LIN {X 0,Y 411.182,Z 344.267,A -85,B 0,C 180,E1 -10470.848,E2 -10470.848} C_VEL
LIN {X 0,Y 411.197,Z 344.265,A -85,B 0,C 180,E1 -10474.334,E2 -10474.334} C_VEL
LIN {X 0,Y 411.18,Z 344.267,A -85,B 0,C 180,E1 -10477.975,E2 -10477.975} C_VEL
LIN {X 0,Y 411.141,Z 344.272,A -85,B 0,C 180,E1 -10481.226,E2 -10481.226} C_VEL
LIN {X 0,Y 411.169,Z 344.265,A -85,B 0,C 180,E1 -10484.492,E2 -10484.492} C_VEL
LIN {X 0,Y 411.213,Z 344.444,A -85,B 0,C 180,E1 -10487.137,E2 -10487.137} C_VEL
LIN {X 0,Y 412.973,Z 353.126,A -85,B 0,C 180,E1 -10490.516,E2 -10490.516} C_VEL
LIN {X 0,Y 414.178,Z 359.884,A -85,B 0,C 180,E1 -10492.894,E2 -10492.894} C_VEL
LIN {X 0,Y 413.948,Z 363.821,A -85,B 0,C 180,E1 -10494.146,E2 -10494.146} C_VEL
LIN {X 0,Y 412.826,Z 377.183,A -85,B 0,C 180,E1 -10498.147,E2 -10498.147} C_VEL
LIN {X 0,Y 412.116,Z 388.901,A -85,B 0,C 180,E1 -10501.479,E2 -10501.479} C_VEL
LIN {X 0,Y 411.506,Z 401.226,A -85,B 0,C 180,E1 -10504.847,E2 -10504.847} C_VEL
LIN {X 0,Y 411.04,Z 414.75,A -85,B 0,C 180,E1 -10508.432,E2 -10508.432} C_VEL
LIN {X 0,Y 410.751,Z 427.741,A -85,B 0,C 180,E1 -10511.805,E2 -10511.805} C_VEL
LIN {X 0,Y 410.736,Z 429.149,A -85,B 0,C 180,E1 -10512.091,E2 -10512.091} C_VEL
LIN {X 0,Y 412.704,Z 446.705,A -85,B 0,C 180,E1 -10512.79,E2 -10512.79} C_VEL
LIN {X 0,Y 413.305,Z 460.605,A -85,B 0,C 180,E1 -10513.516,E2 -10513.516} C_VEL
LIN {X 0,Y 413.672,Z 472.997,A -85,B 0,C 180,E1 -10514.354,E2 -10514.354} C_VEL
LIN {X 0,Y 412.741,Z 484.841,A -85,B 0,C 180,E1 -10515.328,E2 -10515.328} C_VEL
LIN {X 0,Y 411.972,Z 495.807,A -85,B 0,C 180,E1 -10516.46,E2 -10516.46} C_VEL
LIN {X 0,Y 411.62,Z 503.6,A -85,B 0,C 180,E1 -10517.427,E2 -10517.427} C_VEL
LIN {X 0,Y 411.044,Z 512.023,A -85,B 0,C 180,E1 -10518.661,E2 -10518.661} C_VEL
LIN {X 0,Y 410.621,Z 520.378,A -85,B 0,C 180,E1 -10520.145,E2 -10520.145} C_VEL
LIN {X 0,Y 410.458,Z 527.159,A -85,B 0,C 180,E1 -10521.632,E2 -10521.632} C_VEL
LIN {X 0,Y 410.452,Z 533.082,A -85,B 0,C 180,E1 -10523.272,E2 -10523.272} C_VEL
LIN {X 0,Y 410.58,Z 538.034,A -85,B 0,C 180,E1 -10525.09,E2 -10525.09} C_VEL
LIN {X 0,Y 410.673,Z 540.042,A -85,B 0,C 180,E1 -10526.075,E2 -10526.075} C_VEL
LIN {X 0,Y 410.66,Z 542.668,A -85,B 0,C 180,E1 -10528.039,E2 -10528.039} C_VEL
LIN {X 0,Y 410.893,Z 543.399,A -85,B 0,C 180,E1 -10529.02,E2 -10529.02} C_VEL
LIN {X 0,Y 410.904,Z 543.637,A -85,B 0,C 180,E1 -10530,E2 -10530} C_VEL
LIN {X 0,Y 410.886,Z 543.448,A -85,B 0,C 180,E1 -10530.98,E2 -10530.98} C_VEL
LIN {X 0,Y 410.614,Z 541.808,A -85,B 0,C 180,E1 -10532.943,E2 -10532.943} C_VEL
LIN {X 0,Y 410.637,Z 540.321,A -85,B 0,C 180,E1 -10533.925,E2 -10533.925} C_VEL
LIN {X 0,Y 410.505,Z 537.236,A -85,B 0,C 180,E1 -10535.403,E2 -10535.403} C_VEL
LIN {X 0,Y 410.458,Z 533.052,A -85,B 0,C 180,E1 -10536.884,E2 -10536.884} C_VEL
LIN {X 0,Y 410.472,Z 526.635,A -85,B 0,C 180,E1 -10538.616,E2 -10538.616} C_VEL
LIN {X 0,Y 410.643,Z 519.625,A -85,B 0,C 180,E1 -10540.103,E2 -10540.103} C_VEL
LIN {X 0,Y 411.109,Z 510.866,A -85,B 0,C 180,E1 -10541.587,E2 -10541.587} C_VEL
LIN {X 0,Y 411.758,Z 500.837,A -85,B 0,C 180,E1 -10542.962,E2 -10542.962} C_VEL
LIN {X 0,Y 412.365,Z 490.938,A -85,B 0,C 180,E1 -10544.055,E2 -10544.055} C_VEL
LIN {X 0,Y 413.044,Z 479.935,A -85,B 0,C 180,E1 -10545.039,E2 -10545.039} C_VEL
LIN {X 0,Y 413.6,Z 469.683,A -85,B 0,C 180,E1 -10545.776,E2 -10545.776} C_VEL
LIN {X 0,Y 412.83,Z 456.929,A -85,B 0,C 180,E1 -10546.527,E2 -10546.527} C_VEL
LIN {X 0,Y 411.742,Z 444.07,A -85,B 0,C 180,E1 -10547.086,E2 -10547.086} C_VEL
LIN {X 0,Y 410.691,Z 433.86,A -85,B 0,C 180,E1 -10547.445,E2 -10547.445} C_VEL
LIN {X 0,Y 411.003,Z 424.02,A -85,B 0,C 180,E1 -10549.998,E2 -10549.998} C_VEL
LIN {X 0,Y 411.592,Z 410.426,A -85,B 0,C 180,E1 -10553.657,E2 -10553.657} C_VEL
LIN {X 0,Y 412.186,Z 398.684,A -85,B 0,C 180,E1 -10556.861,E2 -10556.861} C_VEL
LIN {X 0,Y 413.082,Z 384.959,A -85,B 0,C 180,E1 -10560.69,E2 -10560.69} C_VEL
LIN {X 0,Y 413.961,Z 373.104,A -85,B 0,C 180,E1 -10564.072,E2 -10564.072} C_VEL
LIN {X 0,Y 414.818,Z 363.878,A -85,B 0,C 180,E1 -10566.78,E2 -10566.78} C_VEL
LIN {X 0,Y 413.734,Z 357.047,A -85,B 0,C 180,E1 -10568.939,E2 -10568.939} C_VEL
LIN {X 0,Y 411.767,Z 347.244,A -85,B 0,C 180,E1 -10572.215,E2 -10572.215} C_VEL
LIN {X 0,Y 411.186,Z 344.328,A -85,B 0,C 180,E1 -10573.299,E2 -10573.299} C_VEL
LIN {X 0,Y 411.159,Z 344.271,A -85,B 0,C 180,E1 -10576.864,E2 -10576.864} C_VEL
LIN {X 0,Y 411.163,Z 344.265,A -85,B 0,C 180,E1 -10580.279,E2 -10580.279} C_VEL
LIN {X 0,Y 411.186,Z 344.268,A -85,B 0,C 180,E1 -10583.447,E2 -10583.447} C_VEL
LIN {X 0,Y 411.2,Z 344.263,A -85,B 0,C 180,E1 -10586.873,E2 -10586.873} C_VEL
LIN {X 0,Y 411.225,Z 344.258,A -85,B 0,C 180,E1 -10590.644,E2 -10590.644} C_VEL
LIN {X 0,Y 411.229,Z 344.259,A -85,B 0,C 180,E1 -10593.618,E2 -10593.618} C_VEL
LIN {X 0,Y 411.187,Z 344.266,A -85,B 0,C 180,E1 -10596.851,E2 -10596.851} C_VEL
LIN {X 0,Y 411.205,Z 344.259,A -85,B 0,C 180,E1 -10600.05,E2 -10600.05} C_VEL
LIN {X 0,Y 411.254,Z 344.26,A -85,B 0,C 180,E1 -10603.131,E2 -10603.131} C_VEL
LIN {X 0,Y 411.296,Z 344.254,A -85,B 0,C 180,E1 -10606.896,E2 -10606.896} C_VEL
LIN {X 0,Y 411.281,Z 344.25,A -85,B 0,C 180,E1 -10610.161,E2 -10610.161} C_VEL
LIN {X 0,Y 411.426,Z 344.236,A -85,B 0,C 180,E1 -10613.132,E2 -10613.132} C_VEL
LIN {X 0,Y 411.296,Z 344.253,A -85,B 0,C 180,E1 -10615.099,E2 -10615.099} C_VEL
LIN {X 0,Y 411.501,Z 344.223,A -85,B 0,C 180,E1 -10618.042,E2 -10618.042} C_VEL
LIN {X 0,Y 411.631,Z 344.207,A -85,B 0,C 180,E1 -10620,E2 -10620} C_VEL
LIN {X 0,Y 411.446,Z 344.235,A -85,B 0,C 180,E1 -10622.937,E2 -10622.937} C_VEL
LIN {X 0,Y 411.448,Z 344.234,A -85,B 0,C 180,E1 -10626.867,E2 -10626.867} C_VEL
LIN {X 0,Y 411.284,Z 344.25,A -85,B 0,C 180,E1 -10629.839,E2 -10629.839} C_VEL
LIN {X 0,Y 411.296,Z 344.25,A -85,B 0,C 180,E1 -10633.104,E2 -10633.104} C_VEL
LIN {X 0,Y 411.249,Z 344.257,A -85,B 0,C 180,E1 -10636.889,E2 -10636.889} C_VEL
LIN {X 0,Y 411.222,Z 344.259,A -85,B 0,C 180,E1 -10639.987,E2 -10639.987} C_VEL
LIN {X 0,Y 411.196,Z 344.261,A -85,B 0,C 180,E1 -10643.148,E2 -10643.148} C_VEL
LIN {X 0,Y 411.23,Z 344.263,A -85,B 0,C 180,E1 -10646.381,E2 -10646.381} C_VEL
LIN {X 0,Y 411.203,Z 344.26,A -85,B 0,C 180,E1 -10649.713,E2 -10649.713} C_VEL
LIN {X 0,Y 411.2,Z 344.26,A -85,B 0,C 180,E1 -10653.156,E2 -10653.156} C_VEL
LIN {X 0,Y 411.189,Z 344.265,A -85,B 0,C 180,E1 -10656.554,E2 -10656.554} C_VEL
LIN {X 0,Y 411.221,Z 344.259,A -85,B 0,C 180,E1 -10659.731,E2 -10659.731} C_VEL
LIN {X 0,Y 411.172,Z 344.263,A -85,B 0,C 180,E1 -10663.134,E2 -10663.134} C_VEL
LIN {X 0,Y 411.169,Z 344.268,A -85,B 0,C 180,E1 -10665.881,E2 -10665.881} C_VEL
LIN {X 0,Y 411.165,Z 344.265,A -85,B 0,C 180,E1 -10668.772,E2 -10668.772} C_VEL
LIN {X 0,Y 411.208,Z 344.263,A -85,B 0,C 180,E1 -10671.831,E2 -10671.831} C_VEL
LIN {X 0,Y 411.209,Z 344.259,A -85,B 0,C 180,E1 -10675.122,E2 -10675.122} C_VEL
LIN {X 0,Y 411.17,Z 344.271,A -85,B 0,C 180,E1 -10678.004,E2 -10678.004} C_VEL
LIN {X 0,Y 411.223,Z 344.259,A -85,B 0,C 180,E1 -10681.411,E2 -10681.411} C_VEL
LIN {X 0,Y 411.236,Z 344.256,A -85,B 0,C 180,E1 -10684.708,E2 -10684.708} C_VEL
LIN {X 0,Y 411.206,Z 344.266,A -85,B 0,C 180,E1 -10687.914,E2 -10687.914} C_VEL
LIN {X 0,Y 411.226,Z 344.257,A -85,B 0,C 180,E1 -10691.052,E2 -10691.052} C_VEL
LIN {X 0,Y 411.265,Z 344.255,A -85,B 0,C 180,E1 -10694.133,E2 -10694.133} C_VEL
LIN {X 0,Y 411.305,Z 344.248,A -85,B 0,C 180,E1 -10697.166,E2 -10697.166} C_VEL
LIN {X 0,Y 411.296,Z 344.25,A -85,B 0,C 180,E1 -10700.162,E2 -10700.162} C_VEL
LIN {X 0,Y 411.464,Z 344.229,A -85,B 0,C 180,E1 -10703.133,E2 -10703.133} C_VEL
LIN {X 0,Y 411.315,Z 344.248,A -85,B 0,C 180,E1 -10705.099,E2 -10705.099} C_VEL
LIN {X 0,Y 411.516,Z 344.223,A -85,B 0,C 180,E1 -10708.043,E2 -10708.043} C_VEL
LIN {X 0,Y 411.645,Z 344.207,A -85,B 0,C 180,E1 -10710,E2 -10710} C_VEL
LIN {X 0,Y 411.469,Z 344.228,A -85,B 0,C 180,E1 -10712.937,E2 -10712.937} C_VEL
LIN {X 0,Y 411.454,Z 344.23,A -85,B 0,C 180,E1 -10716.867,E2 -10716.867} C_VEL
LIN {X 0,Y 411.295,Z 344.251,A -85,B 0,C 180,E1 -10719.838,E2 -10719.838} C_VEL
LIN {X 0,Y 411.284,Z 344.252,A -85,B 0,C 180,E1 -10723.338,E2 -10723.338} C_VEL
LIN {X 0,Y 411.258,Z 344.255,A -85,B 0,C 180,E1 -10726.888,E2 -10726.888} C_VEL
LIN {X 0,Y 411.241,Z 344.255,A -85,B 0,C 180,E1 -10727.603,E2 -10727.603} C_VEL
LIN {X 0,Y 410.582,Z 344.339,A -85,B 0,C 180,E1 -10728.421,E2 -10728.421} C_VEL
LIN {X 0,Y 407.694,Z 344.702,A -85,B 0,C 180,E1 -10729.749,E2 -10729.749} C_VEL
LIN {X 0,Y 405.249,Z 345.006,A -85,B 0,C 180,E1 -10730.822,E2 -10730.822} C_VEL
LIN {X 0,Y 404.213,Z 345.134,A -85,B 0,C 180,E1 -10731.652,E2 -10731.652} C_VEL
LIN {X 0,Y 404.137,Z 345.141,A -85,B 0,C 180,E1 -10731.933,E2 -10731.933} C_VEL
LIN {X 0,Y 404.216,Z 345.136,A -85,B 0,C 180,E1 -10735.296,E2 -10735.296} C_VEL
LIN {X 0,Y 404.195,Z 345.133,A -85,B 0,C 180,E1 -10737.999,E2 -10737.999} C_VEL
LIN {X 0,Y 404.138,Z 345.142,A -85,B 0,C 180,E1 -10741.557,E2 -10741.557} C_VEL
LIN {X 0,Y 404.184,Z 345.141,A -85,B 0,C 180,E1 -10745.015,E2 -10745.015} C_VEL
LIN {X 0,Y 404.162,Z 345.141,A -85,B 0,C 180,E1 -10748.755,E2 -10748.755} C_VEL
LIN {X 0,Y 404.188,Z 345.138,A -85,B 0,C 180,E1 -10751.61,E2 -10751.61} C_VEL
LIN {X 0,Y 404.209,Z 345.153,A -85,B 0,C 180,E1 -10755.21,E2 -10755.21} C_VEL
LIN {X 0,Y 404.325,Z 345.754,A -85,B 0,C 180,E1 -10755.451,E2 -10755.451} C_VEL
LIN {X 0,Y 408.011,Z 358.828,A -85,B 0,C 180,E1 -10756.499,E2 -10756.499} C_VEL
LIN {X 0,Y 408.323,Z 361.622,A -85,B 0,C 180,E1 -10756.724,E2 -10756.724} C_VEL
LIN {X 0,Y 407.662,Z 373.344,A -85,B 0,C 180,E1 -10757.751,E2 -10757.751} C_VEL
LIN {X 0,Y 407.014,Z 384.618,A -85,B 0,C 180,E1 -10758.993,E2 -10758.993} C_VEL
LIN {X 0,Y 406.362,Z 393.566,A -85,B 0,C 180,E1 -10760.215,E2 -10760.215} C_VEL
LIN {X 0,Y 405.727,Z 402.619,A -85,B 0,C 180,E1 -10761.738,E2 -10761.738} C_VEL
LIN {X 0,Y 405.279,Z 409.366,A -85,B 0,C 180,E1 -10763.141,E2 -10763.141} C_VEL
LIN {X 0,Y 404.818,Z 415.329,A -85,B 0,C 180,E1 -10764.68,E2 -10764.68} C_VEL
LIN {X 0,Y 404.473,Z 420.74,A -85,B 0,C 180,E1 -10766.513,E2 -10766.513} C_VEL
LIN {X 0,Y 404.354,Z 422.796,A -85,B 0,C 180,E1 -10767.398,E2 -10767.398} C_VEL
LIN {X 0,Y 404.205,Z 424.944,A -85,B 0,C 180,E1 -10768.559,E2 -10768.559} C_VEL
LIN {X 0,Y 404.076,Z 427.221,A -85,B 0,C 180,E1 -10770.414,E2 -10770.414} C_VEL
LIN {X 0,Y 404.051,Z 428.116,A -85,B 0,C 180,E1 -10772.507,E2 -10772.507} C_VEL
LIN {X 0,Y 404.203,Z 427.536,A -85,B 0,C 180,E1 -10774.235,E2 -10774.235} C_VEL
LIN {X 0,Y 404.37,Z 426.551,A -85,B 0,C 180,E1 -10775.347,E2 -10775.347} C_VEL
LIN {X 0,Y 404.7,Z 424.127,A -85,B 0,C 180,E1 -10776.98,E2 -10776.98} C_VEL
LIN {X 0,Y 405.103,Z 420.487,A -85,B 0,C 180,E1 -10778.634,E2 -10778.634} C_VEL
LIN {X 0,Y 405.592,Z 415.659,A -85,B 0,C 180,E1 -10780.252,E2 -10780.252} C_VEL
LIN {X 0,Y 406.191,Z 409.482,A -85,B 0,C 180,E1 -10781.854,E2 -10781.854} C_VEL
LIN {X 0,Y 406.992,Z 401.579,A -85,B 0,C 180,E1 -10783.446,E2 -10783.446} C_VEL
LIN {X 0,Y 407.751,Z 392.971,A -85,B 0,C 180,E1 -10784.838,E2 -10784.838} C_VEL
LIN {X 0,Y 408.537,Z 383.59,A -85,B 0,C 180,E1 -10786.064,E2 -10786.064} C_VEL
LIN {X 0,Y 409.32,Z 372.302,A -85,B 0,C 180,E1 -10787.241,E2 -10787.241} C_VEL
LIN {X 0,Y 409.803,Z 363.324,A -85,B 0,C 180,E1 -10788,E2 -10788} C_VEL
LIN {X 0,Y 408.216,Z 356.856,A -85,B 0,C 180,E1 -10788.58,E2 -10788.58} C_VEL
LIN {X 0,Y 404.382,Z 345.836,A -85,B 0,C 180,E1 -10789.517,E2 -10789.517} C_VEL
LIN {X 0,Y 404.247,Z 345.165,A -85,B 0,C 180,E1 -10789.735,E2 -10789.735} C_VEL
LIN {X 0,Y 404.391,Z 345.114,A -85,B 0,C 180,E1 -10793.012,E2 -10793.012} C_VEL
LIN {X 0,Y 404.269,Z 345.127,A -85,B 0,C 180,E1 -10795.013,E2 -10795.013} C_VEL
LIN {X 0,Y 404.469,Z 345.103,A -85,B 0,C 180,E1 -10798.009,E2 -10798.009} C_VEL
LIN {X 0,Y 404.6,Z 345.086,A -85,B 0,C 180,E1 -10800,E2 -10800} C_VEL
LIN {X 0,Y 404.404,Z 345.113,A -85,B 0,C 180,E1 -10802.989,E2 -10802.989} C_VEL
LIN {X 0,Y 404.402,Z 345.11,A -85,B 0,C 180,E1 -10805.985,E2 -10805.985} C_VEL
LIN {X 0,Y 404.256,Z 345.131,A -85,B 0,C 180,E1 -10809.002,E2 -10809.002} C_VEL
LIN {X 0,Y 404.246,Z 345.127,A -85,B 0,C 180,E1 -10812.042,E2 -10812.042} C_VEL
LIN {X 0,Y 404.196,Z 345.138,A -85,B 0,C 180,E1 -10815.118,E2 -10815.118} C_VEL
LIN {X 0,Y 404.195,Z 345.131,A -85,B 0,C 180,E1 -10818.239,E2 -10818.239} C_VEL
LIN {X 0,Y 404.129,Z 345.145,A -85,B 0,C 180,E1 -10821.42,E2 -10821.42} C_VEL
LIN {X 0,Y 404.166,Z 345.139,A -85,B 0,C 180,E1 -10824.666,E2 -10824.666} C_VEL
LIN {X 0,Y 404.188,Z 345.137,A -85,B 0,C 180,E1 -10828,E2 -10828} C_VEL
LIN {X 0,Y 404.132,Z 345.144,A -85,B 0,C 180,E1 -10831.558,E2 -10831.558} C_VEL
LIN {X 0,Y 404.177,Z 345.139,A -85,B 0,C 180,E1 -10835.017,E2 -10835.017} C_VEL
LIN {X 0,Y 404.128,Z 345.146,A -85,B 0,C 180,E1 -10838.76,E2 -10838.76} C_VEL
LIN {X 0,Y 404.101,Z 345.148,A -85,B 0,C 180,E1 -10841.598,E2 -10841.598} C_VEL
LIN {X 0,Y 404.139,Z 345.141,A -85,B 0,C 180,E1 -10844.523,E2 -10844.523} C_VEL
LIN {X 0,Y 404.136,Z 345.277,A -85,B 0,C 180,E1 -10846.648,E2 -10846.648} C_VEL
LIN {X 0,Y 405.675,Z 352.683,A -85,B 0,C 180,E1 -10849.665,E2 -10849.665} C_VEL
LIN {X 0,Y 407.127,Z 360.603,A -85,B 0,C 180,E1 -10852.568,E2 -10852.568} C_VEL
LIN {X 0,Y 407.293,Z 363.262,A -85,B 0,C 180,E1 -10853.466,E2 -10853.466} C_VEL
LIN {X 0,Y 405.984,Z 376.465,A -85,B 0,C 180,E1 -10857.546,E2 -10857.546} C_VEL
LIN {X 0,Y 405.07,Z 390.069,A -85,B 0,C 180,E1 -10861.503,E2 -10861.503} C_VEL
LIN {X 0,Y 404.435,Z 402.539,A -85,B 0,C 180,E1 -10864.984,E2 -10864.984} C_VEL
LIN {X 0,Y 403.932,Z 415.783,A -85,B 0,C 180,E1 -10868.57,E2 -10868.57} C_VEL
LIN {X 0,Y 403.696,Z 427.647,A -85,B 0,C 180,E1 -10871.673,E2 -10871.673} C_VEL
LIN {X 0,Y 403.778,Z 429.123,A -85,B 0,C 180,E1 -10871.775,E2 -10871.775} C_VEL
LIN {X 0,Y 405.658,Z 444.216,A -85,B 0,C 180,E1 -10872.376,E2 -10872.376} C_VEL
LIN {X 0,Y 406.334,Z 456.955,A -85,B 0,C 180,E1 -10873.03,E2 -10873.03} C_VEL
LIN {X 0,Y 406.708,Z 468.89,A -85,B 0,C 180,E1 -10873.821,E2 -10873.821} C_VEL
LIN {X 0,Y 406.427,Z 477.034,A -85,B 0,C 180,E1 -10874.453,E2 -10874.453} C_VEL
LIN {X 0,Y 405.517,Z 487.877,A -85,B 0,C 180,E1 -10875.446,E2 -10875.446} C_VEL
LIN {X 0,Y 404.805,Z 498.316,A -85,B 0,C 180,E1 -10876.629,E2 -10876.629} C_VEL
LIN {X 0,Y 404.282,Z 506.25,A -85,B 0,C 180,E1 -10877.705,E2 -10877.705} C_VEL
LIN {X 0,Y 403.738,Z 515.491,A -85,B 0,C 180,E1 -10879.215,E2 -10879.215} C_VEL
LIN {X 0,Y 403.458,Z 523.005,A -85,B 0,C 180,E1 -10880.728,E2 -10880.728} C_VEL
LIN {X 0,Y 403.389,Z 529.931,A -85,B 0,C 180,E1 -10882.492,E2 -10882.492} C_VEL
LIN {X 0,Y 403.423,Z 534.558,A -85,B 0,C 180,E1 -10884,E2 -10884} C_VEL
LIN {X 0,Y 403.57,Z 538.084,A -85,B 0,C 180,E1 -10885.505,E2 -10885.505} C_VEL
LIN {X 0,Y 403.591,Z 540.56,A -85,B 0,C 180,E1 -10887.006,E2 -10887.006} C_VEL
LIN {X 0,Y 403.865,Z 542.397,A -85,B 0,C 180,E1 -10889.003,E2 -10889.003} C_VEL
LIN {X 0,Y 403.881,Z 542.626,A -85,B 0,C 180,E1 -10890,E2 -10890} C_VEL
LIN {X 0,Y 403.859,Z 542.434,A -85,B 0,C 180,E1 -10890.997,E2 -10890.997} C_VEL
LIN {X 0,Y 403.607,Z 541.802,A -85,B 0,C 180,E1 -10891.996,E2 -10891.996} C_VEL
LIN {X 0,Y 403.574,Z 540.774,A -85,B 0,C 180,E1 -10892.995,E2 -10892.995} C_VEL
LIN {X 0,Y 403.599,Z 539.275,A -85,B 0,C 180,E1 -10893.994,E2 -10893.994} C_VEL
LIN {X 0,Y 403.452,Z 536.169,A -85,B 0,C 180,E1 -10895.498,E2 -10895.498} C_VEL
LIN {X 0,Y 403.394,Z 531.961,A -85,B 0,C 180,E1 -10897.005,E2 -10897.005} C_VEL
LIN {X 0,Y 403.399,Z 525.518,A -85,B 0,C 180,E1 -10898.768,E2 -10898.768} C_VEL
LIN {X 0,Y 403.605,Z 518.467,A -85,B 0,C 180,E1 -10900.281,E2 -10900.281} C_VEL
LIN {X 0,Y 404.067,Z 509.668,A -85,B 0,C 180,E1 -10901.792,E2 -10901.792} C_VEL
LIN {X 0,Y 404.678,Z 500.703,A -85,B 0,C 180,E1 -10903.048,E2 -10903.048} C_VEL
LIN {X 0,Y 405.329,Z 490.882,A -85,B 0,C 180,E1 -10904.176,E2 -10904.176} C_VEL
LIN {X 0,Y 406.028,Z 480.092,A -85,B 0,C 180,E1 -10905.177,E2 -10905.177} C_VEL
LIN {X 0,Y 406.589,Z 470.113,A -85,B 0,C 180,E1 -10905.926,E2 -10905.926} C_VEL
LIN {X 0,Y 405.841,Z 456.762,A -85,B 0,C 180,E1 -10906.743,E2 -10906.743} C_VEL
LIN {X 0,Y 404.687,Z 443.338,A -85,B 0,C 180,E1 -10907.348,E2 -10907.348} C_VEL
LIN {X 0,Y 403.637,Z 432.958,A -85,B 0,C 180,E1 -10907.724,E2 -10907.724} C_VEL
LIN {X 0,Y 403.909,Z 424.292,A -85,B 0,C 180,E1 -10910.015,E2 -10910.015} C_VEL
LIN {X 0,Y 404.492,Z 411.382,A -85,B 0,C 180,E1 -10913.554,E2 -10913.554} C_VEL
LIN {X 0,Y 405.101,Z 399.7,A -85,B 0,C 180,E1 -10916.811,E2 -10916.811} C_VEL
LIN {X 0,Y 406.04,Z 385.99,A -85,B 0,C 180,E1 -10920.703,E2 -10920.703} C_VEL
LIN {X 0,Y 407.011,Z 373.626,A -85,B 0,C 180,E1 -10924.312,E2 -10924.312} C_VEL
LIN {X 0,Y 407.843,Z 365.306,A -85,B 0,C 180,E1 -10926.784,E2 -10926.784} C_VEL
LIN {X 0,Y 407.087,Z 360.203,A -85,B 0,C 180,E1 -10928.425,E2 -10928.425} C_VEL
LIN {X 0,Y 405.476,Z 351.908,A -85,B 0,C 180,E1 -10931.195,E2 -10931.195} C_VEL
LIN {X 0,Y 404.123,Z 345.237,A -85,B 0,C 180,E1 -10933.554,E2 -10933.554} C_VEL
LIN {X 0,Y 404.139,Z 345.146,A -85,B 0,C 180,E1 -10936.917,E2 -10936.917} C_VEL
LIN {X 0,Y 404.127,Z 345.142,A -85,B 0,C 180,E1 -10939.95,E2 -10939.95} C_VEL
LIN {X 0,Y 404.128,Z 345.146,A -85,B 0,C 180,E1 -10943.125,E2 -10943.125} C_VEL
LIN {X 0,Y 404.138,Z 345.14,A -85,B 0,C 180,E1 -10946.187,E2 -10946.187} C_VEL
LIN {X 0,Y 404.138,Z 345.142,A -85,B 0,C 180,E1 -10949.714,E2 -10949.714} C_VEL
LIN {X 0,Y 404.188,Z 345.14,A -85,B 0,C 180,E1 -10953.122,E2 -10953.122} C_VEL
LIN {X 0,Y 404.166,Z 345.141,A -85,B 0,C 180,E1 -10955.334,E2 -10955.334} C_VEL
LIN {X 0,Y 404.129,Z 345.143,A -85,B 0,C 180,E1 -10958.58,E2 -10958.58} C_VEL
LIN {X 0,Y 404.195,Z 345.133,A -85,B 0,C 180,E1 -10961.761,E2 -10961.761} C_VEL
LIN {X 0,Y 404.196,Z 345.138,A -85,B 0,C 180,E1 -10964.882,E2 -10964.882} C_VEL
LIN {X 0,Y 404.246,Z 345.126,A -85,B 0,C 180,E1 -10967.958,E2 -10967.958} C_VEL
LIN {X 0,Y 404.256,Z 345.132,A -85,B 0,C 180,E1 -10970.998,E2 -10970.998} C_VEL
LIN {X 0,Y 404.402,Z 345.107,A -85,B 0,C 180,E1 -10974.015,E2 -10974.015} C_VEL
LIN {X 0,Y 404.47,Z 345.099,A -85,B 0,C 180,E1 -10978.008,E2 -10978.008} C_VEL
LIN {X 0,Y 404.6,Z 345.082,A -85,B 0,C 180,E1 -10980,E2 -10980} C_VEL
LIN {X 0,Y 404.404,Z 345.111,A -85,B 0,C 180,E1 -10982.989,E2 -10982.989} C_VEL
LIN {X 0,Y 404.395,Z 345.112,A -85,B 0,C 180,E1 -10986.988,E2 -10986.988} C_VEL
LIN {X 0,Y 404.249,Z 345.127,A -85,B 0,C 180,E1 -10990.012,E2 -10990.012} C_VEL
LIN {X 0,Y 404.258,Z 345.126,A -85,B 0,C 180,E1 -10993.212,E2 -10993.212} C_VEL
LIN {X 0,Y 404.207,Z 345.133,A -85,B 0,C 180,E1 -10997.007,E2 -10997.007} C_VEL
LIN {X 0,Y 404.179,Z 345.14,A -85,B 0,C 180,E1 -11000.351,E2 -11000.351} C_VEL
LIN {X 0,Y 404.162,Z 345.137,A -85,B 0,C 180,E1 -11003.575,E2 -11003.575} C_VEL
LIN {X 0,Y 404.176,Z 345.136,A -85,B 0,C 180,E1 -11005.767,E2 -11005.767} C_VEL
LIN {X 0,Y 404.191,Z 345.136,A -85,B 0,C 180,E1 -11008,E2 -11008} C_VEL
LIN {X 0,Y 404.135,Z 345.14,A -85,B 0,C 180,E1 -11011.559,E2 -11011.559} C_VEL
LIN {X 0,Y 404.179,Z 345.135,A -85,B 0,C 180,E1 -11015.017,E2 -11015.017} C_VEL
LIN {X 0,Y 404.157,Z 345.139,A -85,B 0,C 180,E1 -11018.757,E2 -11018.757} C_VEL
LIN {X 0,Y 404.144,Z 345.14,A -85,B 0,C 180,E1 -11021.605,E2 -11021.605} C_VEL
LIN {X 0,Y 404.142,Z 345.142,A -85,B 0,C 180,E1 -11024.523,E2 -11024.523} C_VEL
LIN {X 0,Y 404.169,Z 345.136,A -85,B 0,C 180,E1 -11027.301,E2 -11027.301} C_VEL
LIN {X 0,Y 404.166,Z 345.142,A -85,B 0,C 180,E1 -11029.956,E2 -11029.956} C_VEL
LIN {X 0,Y 404.137,Z 345.14,A -85,B 0,C 180,E1 -11033.125,E2 -11033.125} C_VEL
LIN {X 0,Y 404.143,Z 345.144,A -85,B 0,C 180,E1 -11036.189,E2 -11036.189} C_VEL
LIN {X 0,Y 404.154,Z 345.142,A -85,B 0,C 180,E1 -11039.716,E2 -11039.716} C_VEL
LIN {X 0,Y 404.195,Z 345.133,A -85,B 0,C 180,E1 -11043.124,E2 -11043.124} C_VEL
LIN {X 0,Y 404.177,Z 345.136,A -85,B 0,C 180,E1 -11045.335,E2 -11045.335} C_VEL
LIN {X 0,Y 404.14,Z 345.14,A -85,B 0,C 180,E1 -11048.581,E2 -11048.581} C_VEL
LIN {X 0,Y 404.212,Z 345.137,A -85,B 0,C 180,E1 -11051.763,E2 -11051.763} C_VEL
LIN {X 0,Y 404.213,Z 345.13,A -85,B 0,C 180,E1 -11054.883,E2 -11054.883} C_VEL
LIN {X 0,Y 404.259,Z 345.129,A -85,B 0,C 180,E1 -11057.959,E2 -11057.959} C_VEL
LIN {X 0,Y 404.436,Z 345.105,A -85,B 0,C 180,E1 -11062.1,E2 -11062.1} C_VEL
LIN {X 0,Y 404.428,Z 345.106,A -85,B 0,C 180,E1 -11064.015,E2 -11064.015} C_VEL
LIN {X 0,Y 404.485,Z 345.099,A -85,B 0,C 180,E1 -11068.009,E2 -11068.009} C_VEL
LIN {X 0,Y 404.614,Z 345.083,A -85,B 0,C 180,E1 -11070,E2 -11070} C_VEL
LIN {X 0,Y 404.426,Z 345.106,A -85,B 0,C 180,E1 -11072.988,E2 -11072.988} C_VEL
LIN {X 0,Y 404.402,Z 345.109,A -85,B 0,C 180,E1 -11076.987,E2 -11076.987} C_VEL
LIN {X 0,Y 404.261,Z 345.126,A -85,B 0,C 180,E1 -11080.011,E2 -11080.011} C_VEL
LIN {X 0,Y 404.268,Z 345.129,A -85,B 0,C 180,E1 -11083.211,E2 -11083.211} C_VEL
LIN {X 0,Y 404.217,Z 345.134,A -85,B 0,C 180,E1 -11087.007,E2 -11087.007} C_VEL
LIN {X 0,Y 404.164,Z 345.137,A -85,B 0,C 180,E1 -11090.351,E2 -11090.351} C_VEL
LIN {X 0,Y 404.137,Z 345.141,A -85,B 0,C 180,E1 -11091.933,E2 -11091.933} C_VEL
LIN {X 0,Y 403.495,Z 345.224,A -85,B 0,C 180,E1 -11092.764,E2 -11092.764} C_VEL
LIN {X 0,Y 400.662,Z 345.573,A -85,B 0,C 180,E1 -11094.116,E2 -11094.116} C_VEL
LIN {X 0,Y 398.251,Z 345.88,A -85,B 0,C 180,E1 -11095.208,E2 -11095.208} C_VEL
LIN {X 0,Y 397.217,Z 346.003,A -85,B 0,C 180,E1 -11096.053,E2 -11096.053} C_VEL
LIN {X 0,Y 397.134,Z 346.012,A -85,B 0,C 180,E1 -11096.338,E2 -11096.338} C_VEL
LIN {X 0,Y 397.121,Z 346.015,A -85,B 0,C 180,E1 -11098.543,E2 -11098.543} C_VEL
LIN {X 0,Y 397.077,Z 346.019,A -85,B 0,C 180,E1 -11102.071,E2 -11102.071} C_VEL
LIN {X 0,Y 397.118,Z 346.016,A -85,B 0,C 180,E1 -11105.503,E2 -11105.503} C_VEL
LIN {X 0,Y 397.135,Z 346.018,A -85,B 0,C 180,E1 -11108.862,E2 -11108.862} C_VEL
LIN {X 0,Y 397.155,Z 346.014,A -85,B 0,C 180,E1 -11112.255,E2 -11112.255} C_VEL
LIN {X 0,Y 397.178,Z 346.191,A -85,B 0,C 180,E1 -11115.099,E2 -11115.099} C_VEL
LIN {X 0,Y 397.461,Z 347.376,A -85,B 0,C 180,E1 -11115.283,E2 -11115.283} C_VEL
LIN {X 0,Y 400.94,Z 359.53,A -85,B 0,C 180,E1 -11116.245,E2 -11116.245} C_VEL
LIN {X 0,Y 401.477,Z 362.107,A -85,B 0,C 180,E1 -11116.467,E2 -11116.467} C_VEL
LIN {X 0,Y 400.803,Z 374.04,A -85,B 0,C 180,E1 -11117.522,E2 -11117.522} C_VEL
LIN {X 0,Y 400.168,Z 384.477,A -85,B 0,C 180,E1 -11118.677,E2 -11118.677} C_VEL
LIN {X 0,Y 399.437,Z 394.465,A -85,B 0,C 180,E1 -11120.043,E2 -11120.043} C_VEL
LIN {X 0,Y 398.762,Z 403.537,A -85,B 0,C 180,E1 -11121.591,E2 -11121.591} C_VEL
LIN {X 0,Y 398.261,Z 410.781,A -85,B 0,C 180,E1 -11123.131,E2 -11123.131} C_VEL
LIN {X 0,Y 397.739,Z 417.469,A -85,B 0,C 180,E1 -11124.951,E2 -11124.951} C_VEL
LIN {X 0,Y 397.408,Z 422.476,A -85,B 0,C 180,E1 -11126.755,E2 -11126.755} C_VEL
LIN {X 0,Y 397.229,Z 425.273,A -85,B 0,C 180,E1 -11128.127,E2 -11128.127} C_VEL
LIN {X 0,Y 397.139,Z 426.826,A -85,B 0,C 180,E1 -11129.123,E2 -11129.123} C_VEL
LIN {X 0,Y 397.052,Z 428.114,A -85,B 0,C 180,E1 -11130.29,E2 -11130.29} C_VEL
LIN {X 0,Y 397.049,Z 429.142,A -85,B 0,C 180,E1 -11132.252,E2 -11132.252} C_VEL
LIN {X 0,Y 397.128,Z 428.909,A -85,B 0,C 180,E1 -11133.741,E2 -11133.741} C_VEL
LIN {X 0,Y 397.263,Z 428.147,A -85,B 0,C 180,E1 -11134.876,E2 -11134.876} C_VEL
LIN {X 0,Y 397.642,Z 425.736,A -85,B 0,C 180,E1 -11136.785,E2 -11136.785} C_VEL
LIN {X 0,Y 398.006,Z 422.894,A -85,B 0,C 180,E1 -11138.234,E2 -11138.234} C_VEL
LIN {X 0,Y 398.49,Z 418.521,A -85,B 0,C 180,E1 -11139.884,E2 -11139.884} C_VEL
LIN {X 0,Y 399.117,Z 412.798,A -85,B 0,C 180,E1 -11141.521,E2 -11141.521} C_VEL
LIN {X 0,Y 399.874,Z 405.515,A -85,B 0,C 180,E1 -11143.142,E2 -11143.142} C_VEL
LIN {X 0,Y 400.626,Z 397.885,A -85,B 0,C 180,E1 -11144.509,E2 -11144.509} C_VEL
LIN {X 0,Y 401.436,Z 388.952,A -85,B 0,C 180,E1 -11145.812,E2 -11145.812} C_VEL
LIN {X 0,Y 402.287,Z 378.837,A -85,B 0,C 180,E1 -11147.001,E2 -11147.001} C_VEL
LIN {X 0,Y 403.017,Z 367.809,A -85,B 0,C 180,E1 -11148.049,E2 -11148.049} C_VEL
LIN {X 0,Y 403.151,Z 364.619,A -85,B 0,C 180,E1 -11148.308,E2 -11148.308} C_VEL
LIN {X 0,Y 400.363,Z 355.085,A -85,B 0,C 180,E1 -11149.189,E2 -11149.189} C_VEL
LIN {X 0,Y 397.302,Z 346.567,A -85,B 0,C 180,E1 -11149.94,E2 -11149.94} C_VEL
LIN {X 0,Y 397.228,Z 346.02,A -85,B 0,C 180,E1 -11150.195,E2 -11150.195} C_VEL
LIN {X 0,Y 397.341,Z 345.993,A -85,B 0,C 180,E1 -11152.888,E2 -11152.888} C_VEL
LIN {X 0,Y 397.241,Z 346.003,A -85,B 0,C 180,E1 -11154.925,E2 -11154.925} C_VEL
LIN {X 0,Y 397.438,Z 345.979,A -85,B 0,C 180,E1 -11157.973,E2 -11157.973} C_VEL
LIN {X 0,Y 397.57,Z 345.962,A -85,B 0,C 180,E1 -11160,E2 -11160} C_VEL
LIN {X 0,Y 397.364,Z 345.991,A -85,B 0,C 180,E1 -11163.042,E2 -11163.042} C_VEL
LIN {X 0,Y 397.353,Z 345.988,A -85,B 0,C 180,E1 -11166.092,E2 -11166.092} C_VEL
LIN {X 0,Y 397.226,Z 346.008,A -85,B 0,C 180,E1 -11169.163,E2 -11169.163} C_VEL
LIN {X 0,Y 397.21,Z 346.004,A -85,B 0,C 180,E1 -11172.258,E2 -11172.258} C_VEL
LIN {X 0,Y 397.169,Z 346.013,A -85,B 0,C 180,E1 -11175.392,E2 -11175.392} C_VEL
LIN {X 0,Y 397.149,Z 346.011,A -85,B 0,C 180,E1 -11178.574,E2 -11178.574} C_VEL
LIN {X 0,Y 397.087,Z 346.021,A -85,B 0,C 180,E1 -11181.819,E2 -11181.819} C_VEL
LIN {X 0,Y 397.145,Z 346.013,A -85,B 0,C 180,E1 -11185.513,E2 -11185.513} C_VEL
LIN {X 0,Y 397.115,Z 346.018,A -85,B 0,C 180,E1 -11188.544,E2 -11188.544} C_VEL
LIN {X 0,Y 397.071,Z 346.023,A -85,B 0,C 180,E1 -11192.072,E2 -11192.072} C_VEL
LIN {X 0,Y 397.112,Z 346.019,A -85,B 0,C 180,E1 -11195.504,E2 -11195.504} C_VEL
LIN {X 0,Y 397.087,Z 346.023,A -85,B 0,C 180,E1 -11198.855,E2 -11198.855} C_VEL
LIN {X 0,Y 397.049,Z 346.029,A -85,B 0,C 180,E1 -11202.27,E2 -11202.27} C_VEL
LIN {X 0,Y 397.109,Z 346.021,A -85,B 0,C 180,E1 -11205.649,E2 -11205.649} C_VEL
LIN {X 0,Y 397.121,Z 346.274,A -85,B 0,C 180,E1 -11206.216,E2 -11206.216} C_VEL
LIN {X 0,Y 398.649,Z 353.577,A -85,B 0,C 180,E1 -11209.295,E2 -11209.295} C_VEL
LIN {X 0,Y 400.071,Z 361.351,A -85,B 0,C 180,E1 -11212.233,E2 -11212.233} C_VEL
LIN {X 0,Y 400.351,Z 364.562,A -85,B 0,C 180,E1 -11213.356,E2 -11213.356} C_VEL
LIN {X 0,Y 398.899,Z 378.496,A -85,B 0,C 180,E1 -11217.746,E2 -11217.746} C_VEL
LIN {X 0,Y 398.153,Z 389.28,A -85,B 0,C 180,E1 -11220.961,E2 -11220.961} C_VEL
LIN {X 0,Y 397.489,Z 401.225,A -85,B 0,C 180,E1 -11224.387,E2 -11224.387} C_VEL
LIN {X 0,Y 396.955,Z 412.884,A -85,B 0,C 180,E1 -11227.626,E2 -11227.626} C_VEL
LIN {X 0,Y 396.642,Z 424.8,A -85,B 0,C 180,E1 -11230.865,E2 -11230.865} C_VEL
LIN {X 0,Y 396.615,Z 426.664,A -85,B 0,C 180,E1 -11231.3,E2 -11231.3} C_VEL
LIN {X 0,Y 398.841,Z 444.546,A -85,B 0,C 180,E1 -11232.074,E2 -11232.074} C_VEL
LIN {X 0,Y 399.47,Z 457.704,A -85,B 0,C 180,E1 -11232.796,E2 -11232.796} C_VEL
LIN {X 0,Y 399.792,Z 470.101,A -85,B 0,C 180,E1 -11233.665,E2 -11233.665} C_VEL
LIN {X 0,Y 399.335,Z 479.303,A -85,B 0,C 180,E1 -11234.432,E2 -11234.432} C_VEL
LIN {X 0,Y 398.382,Z 490.683,A -85,B 0,C 180,E1 -11235.571,E2 -11235.571} C_VEL
LIN {X 0,Y 397.738,Z 500.012,A -85,B 0,C 180,E1 -11236.72,E2 -11236.72} C_VEL
LIN {X 0,Y 396.985,Z 510.201,A -85,B 0,C 180,E1 -11238.253,E2 -11238.253} C_VEL
LIN {X 0,Y 396.465,Z 518.51,A -85,B 0,C 180,E1 -11239.79,E2 -11239.79} C_VEL
LIN {X 0,Y 396.314,Z 525.236,A -85,B 0,C 180,E1 -11241.331,E2 -11241.331} C_VEL
LIN {X 0,Y 396.31,Z 530.645,A -85,B 0,C 180,E1 -11242.869,E2 -11242.869} C_VEL
LIN {X 0,Y 396.358,Z 534.878,A -85,B 0,C 180,E1 -11244.404,E2 -11244.404} C_VEL
LIN {X 0,Y 396.593,Z 538.056,A -85,B 0,C 180,E1 -11245.935,E2 -11245.935} C_VEL
LIN {X 0,Y 396.547,Z 539.567,A -85,B 0,C 180,E1 -11246.952,E2 -11246.952} C_VEL
LIN {X 0,Y 396.837,Z 541.393,A -85,B 0,C 180,E1 -11248.985,E2 -11248.985} C_VEL
LIN {X 0,Y 396.858,Z 541.615,A -85,B 0,C 180,E1 -11250,E2 -11250} C_VEL
LIN {X 0,Y 396.83,Z 541.419,A -85,B 0,C 180,E1 -11251.015,E2 -11251.015} C_VEL
LIN {X 0,Y 396.569,Z 540.779,A -85,B 0,C 180,E1 -11252.031,E2 -11252.031} C_VEL
LIN {X 0,Y 396.535,Z 539.734,A -85,B 0,C 180,E1 -11253.048,E2 -11253.048} C_VEL
LIN {X 0,Y 396.562,Z 538.23,A -85,B 0,C 180,E1 -11254.065,E2 -11254.065} C_VEL
LIN {X 0,Y 396.381,Z 535.098,A -85,B 0,C 180,E1 -11255.596,E2 -11255.596} C_VEL
LIN {X 0,Y 396.312,Z 530.863,A -85,B 0,C 180,E1 -11257.131,E2 -11257.131} C_VEL
LIN {X 0,Y 396.327,Z 525.406,A -85,B 0,C 180,E1 -11258.669,E2 -11258.669} C_VEL
LIN {X 0,Y 396.49,Z 518.566,A -85,B 0,C 180,E1 -11260.21,E2 -11260.21} C_VEL
LIN {X 0,Y 396.97,Z 510.063,A -85,B 0,C 180,E1 -11261.747,E2 -11261.747} C_VEL
LIN {X 0,Y 397.604,Z 501.36,A -85,B 0,C 180,E1 -11263.024,E2 -11263.024} C_VEL
LIN {X 0,Y 398.088,Z 493.34,A -85,B 0,C 180,E1 -11264.01,E2 -11264.01} C_VEL
LIN {X 0,Y 398.926,Z 481.572,A -85,B 0,C 180,E1 -11265.192,E2 -11265.192} C_VEL
LIN {X 0,Y 399.622,Z 472.153,A -85,B 0,C 180,E1 -11265.949,E2 -11265.949} C_VEL
LIN {X 0,Y 399.027,Z 459.899,A -85,B 0,C 180,E1 -11266.77,E2 -11266.77} C_VEL
LIN {X 0,Y 398.021,Z 446.752,A -85,B 0,C 180,E1 -11267.437,E2 -11267.437} C_VEL
LIN {X 0,Y 396.567,Z 431.994,A -85,B 0,C 180,E1 -11268.014,E2 -11268.014} C_VEL
LIN {X 0,Y 396.908,Z 421.987,A -85,B 0,C 180,E1 -11270.74,E2 -11270.74} C_VEL
LIN {X 0,Y 397.494,Z 410.396,A -85,B 0,C 180,E1 -11273.994,E2 -11273.994} C_VEL
LIN {X 0,Y 398.238,Z 397.386,A -85,B 0,C 180,E1 -11277.704,E2 -11277.704} C_VEL
LIN {X 0,Y 399.157,Z 385.054,A -85,B 0,C 180,E1 -11281.292,E2 -11281.292} C_VEL
LIN {X 0,Y 400.14,Z 373.229,A -85,B 0,C 180,E1 -11284.814,E2 -11284.814} C_VEL
LIN {X 0,Y 400.855,Z 367.376,A -85,B 0,C 180,E1 -11286.59,E2 -11286.59} C_VEL
LIN {X 0,Y 400.496,Z 363.335,A -85,B 0,C 180,E1 -11287.892,E2 -11287.892} C_VEL
LIN {X 0,Y 398.876,Z 354.857,A -85,B 0,C 180,E1 -11290.743,E2 -11290.743} C_VEL
LIN {X 0,Y 397.107,Z 346.106,A -85,B 0,C 180,E1 -11293.883,E2 -11293.883} C_VEL
LIN {X 0,Y 397.093,Z 346.022,A -85,B 0,C 180,E1 -11296.521,E2 -11296.521} C_VEL
LIN {X 0,Y 397.08,Z 346.019,A -85,B 0,C 180,E1 -11300.419,E2 -11300.419} C_VEL
LIN {X 0,Y 397.09,Z 346.021,A -85,B 0,C 180,E1 -11303.004,E2 -11303.004} C_VEL
LIN {X 0,Y 397.111,Z 346.015,A -85,B 0,C 180,E1 -11306.282,E2 -11306.282} C_VEL
LIN {X 0,Y 397.098,Z 346.017,A -85,B 0,C 180,E1 -11310.135,E2 -11310.135} C_VEL
LIN {X 0,Y 397.187,Z 346.007,A -85,B 0,C 180,E1 -11312.609,E2 -11312.609} C_VEL
LIN {X 0,Y 397.12,Z 346.014,A -85,B 0,C 180,E1 -11315.981,E2 -11315.981} C_VEL
LIN {X 0,Y 397.13,Z 346.014,A -85,B 0,C 180,E1 -11319.704,E2 -11319.704} C_VEL
LIN {X 0,Y 397.173,Z 346.012,A -85,B 0,C 180,E1 -11322.845,E2 -11322.845} C_VEL
LIN {X 0,Y 397.22,Z 346.005,A -85,B 0,C 180,E1 -11326.702,E2 -11326.702} C_VEL
LIN {X 0,Y 397.207,Z 346.003,A -85,B 0,C 180,E1 -11329.809,E2 -11329.809} C_VEL
LIN {X 0,Y 397.324,Z 345.996,A -85,B 0,C 180,E1 -11332.887,E2 -11332.887} C_VEL
LIN {X 0,Y 397.24,Z 346.006,A -85,B 0,C 180,E1 -11334.925,E2 -11334.925} C_VEL
LIN {X 0,Y 397.439,Z 345.974,A -85,B 0,C 180,E1 -11337.973,E2 -11337.973} C_VEL
LIN {X 0,Y 397.57,Z 345.958,A -85,B 0,C 180,E1 -11340,E2 -11340} C_VEL
LIN {X 0,Y 397.363,Z 345.988,A -85,B 0,C 180,E1 -11343.042,E2 -11343.042} C_VEL
LIN {X 0,Y 397.336,Z 345.987,A -85,B 0,C 180,E1 -11346.707,E2 -11346.707} C_VEL
LIN {X 0,Y 397.243,Z 346.001,A -85,B 0,C 180,E1 -11349.162,E2 -11349.162} C_VEL
LIN {X 0,Y 397.21,Z 346.006,A -85,B 0,C 180,E1 -11352.258,E2 -11352.258} C_VEL
LIN {X 0,Y 397.17,Z 346.008,A -85,B 0,C 180,E1 -11355.392,E2 -11355.392} C_VEL
LIN {X 0,Y 397.154,Z 346.017,A -85,B 0,C 180,E1 -11358.574,E2 -11358.574} C_VEL
LIN {X 0,Y 397.09,Z 346.019,A -85,B 0,C 180,E1 -11361.819,E2 -11361.819} C_VEL
LIN {X 0,Y 397.149,Z 346.011,A -85,B 0,C 180,E1 -11365.132,E2 -11365.132} C_VEL
LIN {X 0,Y 397.156,Z 346.01,A -85,B 0,C 180,E1 -11367.777,E2 -11367.777} C_VEL
LIN {X 0,Y 397.077,Z 346.021,A -85,B 0,C 180,E1 -11370.883,E2 -11370.883} C_VEL
LIN {X 0,Y 397.119,Z 346.019,A -85,B 0,C 180,E1 -11374.494,E2 -11374.494} C_VEL
LIN {X 0,Y 397.103,Z 346.023,A -85,B 0,C 180,E1 -11378.275,E2 -11378.275} C_VEL
LIN {X 0,Y 397.107,Z 346.016,A -85,B 0,C 180,E1 -11380.907,E2 -11380.907} C_VEL
LIN {X 0,Y 397.098,Z 346.018,A -85,B 0,C 180,E1 -11383.649,E2 -11383.649} C_VEL
LIN {X 0,Y 397.103,Z 346.019,A -85,B 0,C 180,E1 -11386.521,E2 -11386.521} C_VEL
LIN {X 0,Y 397.112,Z 346.018,A -85,B 0,C 180,E1 -11390.424,E2 -11390.424} C_VEL
LIN {X 0,Y 397.107,Z 346.02,A -85,B 0,C 180,E1 -11394.266,E2 -11394.266} C_VEL
LIN {X 0,Y 397.113,Z 346.015,A -85,B 0,C 180,E1 -11396.728,E2 -11396.728} C_VEL
LIN {X 0,Y 397.133,Z 346.016,A -85,B 0,C 180,E1 -11400.297,E2 -11400.297} C_VEL
LIN {X 0,Y 397.194,Z 346.005,A -85,B 0,C 180,E1 -11402.611,E2 -11402.611} C_VEL
LIN {X 0,Y 397.133,Z 346.018,A -85,B 0,C 180,E1 -11405.982,E2 -11405.982} C_VEL
LIN {X 0,Y 397.139,Z 346.017,A -85,B 0,C 180,E1 -11409.705,E2 -11409.705} C_VEL
LIN {X 0,Y 397.185,Z 346.006,A -85,B 0,C 180,E1 -11412.844,E2 -11412.844} C_VEL
LIN {X 0,Y 397.181,Z 346.013,A -85,B 0,C 180,E1 -11415.657,E2 -11415.657} C_VEL
LIN {X 0,Y 397.201,Z 346.004,A -85,B 0,C 180,E1 -11418.777,E2 -11418.777} C_VEL
LIN {X 0,Y 397.397,Z 345.982,A -85,B 0,C 180,E1 -11422.041,E2 -11422.041} C_VEL
LIN {X 0,Y 397.259,Z 345.997,A -85,B 0,C 180,E1 -11424.925,E2 -11424.925} C_VEL
LIN {X 0,Y 397.454,Z 345.975,A -85,B 0,C 180,E1 -11427.973,E2 -11427.973} C_VEL
LIN {X 0,Y 397.584,Z 345.958,A -85,B 0,C 180,E1 -11430,E2 -11430} C_VEL
LIN {X 0,Y 397.384,Z 345.983,A -85,B 0,C 180,E1 -11433.041,E2 -11433.041} C_VEL
LIN {X 0,Y 397.373,Z 345.984,A -85,B 0,C 180,E1 -11436.091,E2 -11436.091} C_VEL
LIN {X 0,Y 397.255,Z 346.001,A -85,B 0,C 180,E1 -11439.162,E2 -11439.162} C_VEL
LIN {X 0,Y 397.221,Z 346.001,A -85,B 0,C 180,E1 -11442.258,E2 -11442.258} C_VEL
LIN {X 0,Y 397.181,Z 346.013,A -85,B 0,C 180,E1 -11445.392,E2 -11445.392} C_VEL
LIN {X 0,Y 397.164,Z 346.009,A -85,B 0,C 180,E1 -11448.573,E2 -11448.573} C_VEL
LIN {X 0,Y 397.092,Z 346.018,A -85,B 0,C 180,E1 -11451.927,E2 -11451.927} C_VEL
LIN {X 0,Y 397.153,Z 346.013,A -85,B 0,C 180,E1 -11455.512,E2 -11455.512} C_VEL
LIN {X 0,Y 397.134,Z 346.012,A -85,B 0,C 180,E1 -11456.338,E2 -11456.338} C_VEL
LIN {X 0,Y 396.465,Z 346.103,A -85,B 0,C 180,E1 -11457.185,E2 -11457.185} C_VEL
LIN {X 0,Y 393.589,Z 346.455,A -85,B 0,C 180,E1 -11458.56,E2 -11458.56} C_VEL
LIN {X 0,Y 391.15,Z 346.759,A -85,B 0,C 180,E1 -11459.672,E2 -11459.672} C_VEL
LIN {X 0,Y 390.098,Z 346.89,A -85,B 0,C 180,E1 -11460.532,E2 -11460.532} C_VEL
LIN {X 0,Y 390.01,Z 346.898,A -85,B 0,C 180,E1 -11460.823,E2 -11460.823} C_VEL
LIN {X 0,Y 390.066,Z 346.893,A -85,B 0,C 180,E1 -11464.024,E2 -11464.024} C_VEL
LIN {X 0,Y 390.045,Z 346.897,A -85,B 0,C 180,E1 -11467.551,E2 -11467.551} C_VEL
LIN {X 0,Y 390.08,Z 346.898,A -85,B 0,C 180,E1 -11470.825,E2 -11470.825} C_VEL
LIN {X 0,Y 390.124,Z 346.89,A -85,B 0,C 180,E1 -11473.897,E2 -11473.897} C_VEL
LIN {X 0,Y 390.137,Z 347.093,A -85,B 0,C 180,E1 -11474.848,E2 -11474.848} C_VEL
LIN {X 0,Y 390.42,Z 348.247,A -85,B 0,C 180,E1 -11475.024,E2 -11475.024} C_VEL
LIN {X 0,Y 393.657,Z 359.675,A -85,B 0,C 180,E1 -11475.936,E2 -11475.936} C_VEL
LIN {X 0,Y 394.607,Z 363.325,A -85,B 0,C 180,E1 -11476.263,E2 -11476.263} C_VEL
LIN {X 0,Y 393.902,Z 374.963,A -85,B 0,C 180,E1 -11477.313,E2 -11477.313} C_VEL
LIN {X 0,Y 393.185,Z 386.296,A -85,B 0,C 180,E1 -11478.596,E2 -11478.596} C_VEL
LIN {X 0,Y 392.517,Z 395.325,A -85,B 0,C 180,E1 -11479.866,E2 -11479.866} C_VEL
LIN {X 0,Y 391.815,Z 404.258,A -85,B 0,C 180,E1 -11481.41,E2 -11481.41} C_VEL
LIN {X 0,Y 391.272,Z 411.692,A -85,B 0,C 180,E1 -11483.006,E2 -11483.006} C_VEL
LIN {X 0,Y 390.744,Z 418.406,A -85,B 0,C 180,E1 -11484.861,E2 -11484.861} C_VEL
LIN {X 0,Y 390.395,Z 423.44,A -85,B 0,C 180,E1 -11486.697,E2 -11486.697} C_VEL
LIN {X 0,Y 390.176,Z 426.928,A -85,B 0,C 180,E1 -11488.509,E2 -11488.509} C_VEL
LIN {X 0,Y 390.052,Z 428.728,A -85,B 0,C 180,E1 -11489.865,E2 -11489.865} C_VEL
LIN {X 0,Y 390.017,Z 429.582,A -85,B 0,C 180,E1 -11490.887,E2 -11490.887} C_VEL
LIN {X 0,Y 390.016,Z 430.108,A -85,B 0,C 180,E1 -11492.062,E2 -11492.062} C_VEL
LIN {X 0,Y 390.083,Z 430.13,A -85,B 0,C 180,E1 -11493.229,E2 -11493.229} C_VEL
LIN {X 0,Y 390.196,Z 429.624,A -85,B 0,C 180,E1 -11494.388,E2 -11494.388} C_VEL
LIN {X 0,Y 390.38,Z 428.663,A -85,B 0,C 180,E1 -11495.539,E2 -11495.539} C_VEL
LIN {X 0,Y 390.627,Z 427.148,A -85,B 0,C 180,E1 -11496.683,E2 -11496.683} C_VEL
LIN {X 0,Y 391.075,Z 423.969,A -85,B 0,C 180,E1 -11498.383,E2 -11498.383} C_VEL
LIN {X 0,Y 391.574,Z 419.611,A -85,B 0,C 180,E1 -11500.061,E2 -11500.061} C_VEL
LIN {X 0,Y 392.336,Z 413.208,A -85,B 0,C 180,E1 -11501.896,E2 -11501.896} C_VEL
LIN {X 0,Y 393.072,Z 406.633,A -85,B 0,C 180,E1 -11503.377,E2 -11503.377} C_VEL
LIN {X 0,Y 393.959,Z 398.183,A -85,B 0,C 180,E1 -11504.911,E2 -11504.911} C_VEL
LIN {X 0,Y 394.859,Z 389.09,A -85,B 0,C 180,E1 -11506.228,E2 -11506.228} C_VEL
LIN {X 0,Y 395.703,Z 378.618,A -85,B 0,C 180,E1 -11507.46,E2 -11507.46} C_VEL
LIN {X 0,Y 396.47,Z 367.529,A -85,B 0,C 180,E1 -11508.497,E2 -11508.497} C_VEL
LIN {X 0,Y 396.128,Z 364.838,A -85,B 0,C 180,E1 -11508.746,E2 -11508.746} C_VEL
LIN {X 0,Y 392.836,Z 354.528,A -85,B 0,C 180,E1 -11509.72,E2 -11509.72} C_VEL
LIN {X 0,Y 390.282,Z 347.559,A -85,B 0,C 180,E1 -11510.346,E2 -11510.346} C_VEL
LIN {X 0,Y 390.183,Z 346.906,A -85,B 0,C 180,E1 -11510.605,E2 -11510.605} C_VEL
LIN {X 0,Y 390.293,Z 346.871,A -85,B 0,C 180,E1 -11512.759,E2 -11512.759} C_VEL
LIN {X 0,Y 390.213,Z 346.878,A -85,B 0,C 180,E1 -11514.833,E2 -11514.833} C_VEL
LIN {X 0,Y 390.407,Z 346.855,A -85,B 0,C 180,E1 -11517.937,E2 -11517.937} C_VEL
LIN {X 0,Y 390.539,Z 346.838,A -85,B 0,C 180,E1 -11520,E2 -11520} C_VEL
LIN {X 0,Y 390.299,Z 346.87,A -85,B 0,C 180,E1 -11523.097,E2 -11523.097} C_VEL
LIN {X 0,Y 390.306,Z 346.865,A -85,B 0,C 180,E1 -11526.202,E2 -11526.202} C_VEL
LIN {X 0,Y 390.184,Z 346.883,A -85,B 0,C 180,E1 -11529.329,E2 -11529.329} C_VEL
LIN {X 0,Y 390.161,Z 346.883,A -85,B 0,C 180,E1 -11532.483,E2 -11532.483} C_VEL
LIN {X 0,Y 390.13,Z 346.889,A -85,B 0,C 180,E1 -11535.677,E2 -11535.677} C_VEL
LIN {X 0,Y 390.094,Z 346.893,A -85,B 0,C 180,E1 -11538.923,E2 -11538.923} C_VEL
LIN {X 0,Y 390.029,Z 346.901,A -85,B 0,C 180,E1 -11542.235,E2 -11542.235} C_VEL
LIN {X 0,Y 390.111,Z 346.888,A -85,B 0,C 180,E1 -11545.744,E2 -11545.744} C_VEL
LIN {X 0,Y 390.051,Z 346.897,A -85,B 0,C 180,E1 -11549.11,E2 -11549.11} C_VEL
LIN {X 0,Y 390.036,Z 346.902,A -85,B 0,C 180,E1 -11552.722,E2 -11552.722} C_VEL
LIN {X 0,Y 390.049,Z 346.899,A -85,B 0,C 180,E1 -11555.826,E2 -11555.826} C_VEL
LIN {X 0,Y 390.031,Z 346.904,A -85,B 0,C 180,E1 -11559.213,E2 -11559.213} C_VEL
LIN {X 0,Y 390.025,Z 346.904,A -85,B 0,C 180,E1 -11562.373,E2 -11562.373} C_VEL
LIN {X 0,Y 390.091,Z 347.102,A -85,B 0,C 180,E1 -11565.685,E2 -11565.685} C_VEL
LIN {X 0,Y 391.593,Z 354.518,A -85,B 0,C 180,E1 -11568.919,E2 -11568.919} C_VEL
LIN {X 0,Y 393.022,Z 362.102,A -85,B 0,C 180,E1 -11571.888,E2 -11571.888} C_VEL
LIN {X 0,Y 393.416,Z 365.567,A -85,B 0,C 180,E1 -11573.137,E2 -11573.137} C_VEL
LIN {X 0,Y 392.006,Z 378.787,A -85,B 0,C 180,E1 -11577.419,E2 -11577.419} C_VEL
LIN {X 0,Y 391.119,Z 390.455,A -85,B 0,C 180,E1 -11580.978,E2 -11580.978} C_VEL
LIN {X 0,Y 390.414,Z 402.145,A -85,B 0,C 180,E1 -11584.404,E2 -11584.404} C_VEL
LIN {X 0,Y 389.864,Z 413.94,A -85,B 0,C 180,E1 -11587.756,E2 -11587.756} C_VEL
LIN {X 0,Y 389.564,Z 425.234,A -85,B 0,C 180,E1 -11590.846,E2 -11590.846} C_VEL
LIN {X 0,Y 389.755,Z 427.199,A -85,B 0,C 180,E1 -11590.97,E2 -11590.97} C_VEL
LIN {X 0,Y 391.553,Z 440.056,A -85,B 0,C 180,E1 -11591.52,E2 -11591.52} C_VEL
LIN {X 0,Y 392.483,Z 452.655,A -85,B 0,C 180,E1 -11592.193,E2 -11592.193} C_VEL
LIN {X 0,Y 392.737,Z 466.136,A -85,B 0,C 180,E1 -11593.095,E2 -11593.095} C_VEL
LIN {X 0,Y 392.725,Z 475.861,A -85,B 0,C 180,E1 -11593.897,E2 -11593.897} C_VEL
LIN {X 0,Y 391.614,Z 487.615,A -85,B 0,C 180,E1 -11595.05,E2 -11595.05} C_VEL
LIN {X 0,Y 390.772,Z 497.259,A -85,B 0,C 180,E1 -11596.213,E2 -11596.213} C_VEL
LIN {X 0,Y 390.367,Z 504.545,A -85,B 0,C 180,E1 -11597.259,E2 -11597.259} C_VEL
LIN {X 0,Y 389.719,Z 513.699,A -85,B 0,C 180,E1 -11598.822,E2 -11598.822} C_VEL
LIN {X 0,Y 389.332,Z 521.112,A -85,B 0,C 180,E1 -11600.388,E2 -11600.388} C_VEL
LIN {X 0,Y 389.227,Z 528.011,A -85,B 0,C 180,E1 -11602.217,E2 -11602.217} C_VEL
LIN {X 0,Y 389.3,Z 532.621,A -85,B 0,C 180,E1 -11603.782,E2 -11603.782} C_VEL
LIN {X 0,Y 389.34,Z 535.09,A -85,B 0,C 180,E1 -11604.822,E2 -11604.822} C_VEL
LIN {X 0,Y 389.527,Z 537.066,A -85,B 0,C 180,E1 -11605.862,E2 -11605.862} C_VEL
LIN {X 0,Y 389.503,Z 538.577,A -85,B 0,C 180,E1 -11606.897,E2 -11606.897} C_VEL
LIN {X 0,Y 389.535,Z 539.682,A -85,B 0,C 180,E1 -11607.932,E2 -11607.932} C_VEL
LIN {X 0,Y 389.807,Z 540.384,A -85,B 0,C 180,E1 -11608.967,E2 -11608.967} C_VEL
LIN {X 0,Y 389.835,Z 540.596,A -85,B 0,C 180,E1 -11610,E2 -11610} C_VEL
LIN {X 0,Y 389.801,Z 540.39,A -85,B 0,C 180,E1 -11611.033,E2 -11611.033} C_VEL
LIN {X 0,Y 389.533,Z 539.743,A -85,B 0,C 180,E1 -11612.068,E2 -11612.068} C_VEL
LIN {X 0,Y 389.498,Z 538.672,A -85,B 0,C 180,E1 -11613.103,E2 -11613.103} C_VEL
LIN {X 0,Y 389.523,Z 537.154,A -85,B 0,C 180,E1 -11614.139,E2 -11614.139} C_VEL
LIN {X 0,Y 389.34,Z 533.994,A -85,B 0,C 180,E1 -11615.698,E2 -11615.698} C_VEL
LIN {X 0,Y 389.255,Z 529.724,A -85,B 0,C 180,E1 -11617.261,E2 -11617.261} C_VEL
LIN {X 0,Y 389.276,Z 523.211,A -85,B 0,C 180,E1 -11619.089,E2 -11619.089} C_VEL
LIN {X 0,Y 389.533,Z 516.044,A -85,B 0,C 180,E1 -11620.657,E2 -11620.657} C_VEL
LIN {X 0,Y 390.009,Z 507.144,A -85,B 0,C 180,E1 -11622.224,E2 -11622.224} C_VEL
LIN {X 0,Y 390.545,Z 500.001,A -85,B 0,C 180,E1 -11623.264,E2 -11623.264} C_VEL
LIN {X 0,Y 391.32,Z 489.281,A -85,B 0,C 180,E1 -11624.562,E2 -11624.562} C_VEL
LIN {X 0,Y 392.179,Z 478.608,A -85,B 0,C 180,E1 -11625.593,E2 -11625.593} C_VEL
LIN {X 0,Y 392.524,Z 470.509,A -85,B 0,C 180,E1 -11626.245,E2 -11626.245} C_VEL
LIN {X 0,Y 391.948,Z 458.791,A -85,B 0,C 180,E1 -11627.038,E2 -11627.038} C_VEL
LIN {X 0,Y 390.891,Z 445.227,A -85,B 0,C 180,E1 -11627.737,E2 -11627.737} C_VEL
LIN {X 0,Y 389.543,Z 431.316,A -85,B 0,C 180,E1 -11628.268,E2 -11628.268} C_VEL
LIN {X 0,Y 389.751,Z 424.78,A -85,B 0,C 180,E1 -11630.035,E2 -11630.035} C_VEL
LIN {X 0,Y 390.395,Z 411.294,A -85,B 0,C 180,E1 -11633.894,E2 -11633.894} C_VEL
LIN {X 0,Y 391.064,Z 399.684,A -85,B 0,C 180,E1 -11637.275,E2 -11637.275} C_VEL
LIN {X 0,Y 392.124,Z 386.058,A -85,B 0,C 180,E1 -11641.316,E2 -11641.316} C_VEL
LIN {X 0,Y 393.359,Z 372.338,A -85,B 0,C 180,E1 -11645.496,E2 -11645.496} C_VEL
LIN {X 0,Y 393.863,Z 367.792,A -85,B 0,C 180,E1 -11646.909,E2 -11646.909} C_VEL
LIN {X 0,Y 393.088,Z 362.272,A -85,B 0,C 180,E1 -11648.737,E2 -11648.737} C_VEL
LIN {X 0,Y 391.188,Z 352.724,A -85,B 0,C 180,E1 -11652.074,E2 -11652.074} C_VEL
LIN {X 0,Y 390.068,Z 346.981,A -85,B 0,C 180,E1 -11654.209,E2 -11654.209} C_VEL
LIN {X 0,Y 390.026,Z 346.903,A -85,B 0,C 180,E1 -11657.627,E2 -11657.627} C_VEL
LIN {X 0,Y 390.052,Z 346.897,A -85,B 0,C 180,E1 -11660.903,E2 -11660.903} C_VEL
LIN {X 0,Y 390.078,Z 346.893,A -85,B 0,C 180,E1 -11664.792,E2 -11664.792} C_VEL
LIN {X 0,Y 390.016,Z 346.899,A -85,B 0,C 180,E1 -11668.495,E2 -11668.495} C_VEL
LIN {X 0,Y 390.111,Z 346.887,A -85,B 0,C 180,E1 -11672.069,E2 -11672.069} C_VEL
LIN {X 0,Y 390.069,Z 346.895,A -85,B 0,C 180,E1 -11675.518,E2 -11675.518} C_VEL
LIN {X 0,Y 390.079,Z 346.893,A -85,B 0,C 180,E1 -11679.53,E2 -11679.53} C_VEL
LIN {X 0,Y 390.129,Z 346.889,A -85,B 0,C 180,E1 -11683.248,E2 -11683.248} C_VEL
LIN {X 0,Y 390.186,Z 346.88,A -85,B 0,C 180,E1 -11686.561,E2 -11686.561} C_VEL
LIN {X 0,Y 390.158,Z 346.882,A -85,B 0,C 180,E1 -11689.622,E2 -11689.622} C_VEL
LIN {X 0,Y 390.271,Z 346.872,A -85,B 0,C 180,E1 -11692.758,E2 -11692.758} C_VEL
LIN {X 0,Y 390.211,Z 346.881,A -85,B 0,C 180,E1 -11694.833,E2 -11694.833} C_VEL
LIN {X 0,Y 390.408,Z 346.85,A -85,B 0,C 180,E1 -11697.937,E2 -11697.937} C_VEL
LIN {X 0,Y 390.539,Z 346.834,A -85,B 0,C 180,E1 -11700,E2 -11700} C_VEL
LIN {X 0,Y 390.298,Z 346.867,A -85,B 0,C 180,E1 -11703.097,E2 -11703.097} C_VEL
LIN {X 0,Y 390.29,Z 346.864,A -85,B 0,C 180,E1 -11706.703,E2 -11706.703} C_VEL
LIN {X 0,Y 390.196,Z 346.877,A -85,B 0,C 180,E1 -11709.329,E2 -11709.329} C_VEL
LIN {X 0,Y 390.186,Z 346.878,A -85,B 0,C 180,E1 -11713.439,E2 -11713.439} C_VEL
LIN {X 0,Y 390.14,Z 346.884,A -85,B 0,C 180,E1 -11717.308,E2 -11717.308} C_VEL
LIN {X 0,Y 390.085,Z 346.897,A -85,B 0,C 180,E1 -11720.473,E2 -11720.473} C_VEL
LIN {X 0,Y 390.082,Z 346.891,A -85,B 0,C 180,E1 -11723.351,E2 -11723.351} C_VEL
LIN {X 0,Y 390.106,Z 346.891,A -85,B 0,C 180,E1 -11726.769,E2 -11726.769} C_VEL
LIN {X 0,Y 390.037,Z 346.903,A -85,B 0,C 180,E1 -11730.3,E2 -11730.3} C_VEL
LIN {X 0,Y 390.062,Z 346.897,A -85,B 0,C 180,E1 -11734.025,E2 -11734.025} C_VEL
LIN {X 0,Y 390.041,Z 346.896,A -85,B 0,C 180,E1 -11737.552,E2 -11737.552} C_VEL
LIN {X 0,Y 390.072,Z 346.893,A -85,B 0,C 180,E1 -11740.826,E2 -11740.826} C_VEL
LIN {X 0,Y 390.051,Z 346.898,A -85,B 0,C 180,E1 -11743.887,E2 -11743.887} C_VEL
LIN {X 0,Y 390.06,Z 346.895,A -85,B 0,C 180,E1 -11747.623,E2 -11747.623} C_VEL
LIN {X 0,Y 390.089,Z 346.89,A -85,B 0,C 180,E1 -11750.909,E2 -11750.909} C_VEL
LIN {X 0,Y 390.084,Z 346.891,A -85,B 0,C 180,E1 -11754.794,E2 -11754.794} C_VEL
LIN {X 0,Y 390.046,Z 346.897,A -85,B 0,C 180,E1 -11758.499,E2 -11758.499} C_VEL
LIN {X 0,Y 390.116,Z 346.892,A -85,B 0,C 180,E1 -11762.071,E2 -11762.071} C_VEL
LIN {X 0,Y 390.08,Z 346.894,A -85,B 0,C 180,E1 -11765.52,E2 -11765.52} C_VEL
LIN {X 0,Y 390.056,Z 346.894,A -85,B 0,C 180,E1 -11768.878,E2 -11768.878} C_VEL
LIN {X 0,Y 390.13,Z 346.888,A -85,B 0,C 180,E1 -11772.167,E2 -11772.167} C_VEL
LIN {X 0,Y 390.149,Z 346.885,A -85,B 0,C 180,E1 -11775.393,E2 -11775.393} C_VEL
LIN {X 0,Y 390.15,Z 346.882,A -85,B 0,C 180,E1 -11778.572,E2 -11778.572} C_VEL
LIN {X 0,Y 390.346,Z 346.861,A -85,B 0,C 180,E1 -11781.993,E2 -11781.993} C_VEL
LIN {X 0,Y 390.23,Z 346.873,A -85,B 0,C 180,E1 -11784.834,E2 -11784.834} C_VEL
LIN {X 0,Y 390.423,Z 346.851,A -85,B 0,C 180,E1 -11787.937,E2 -11787.937} C_VEL
LIN {X 0,Y 390.553,Z 346.834,A -85,B 0,C 180,E1 -11790,E2 -11790} C_VEL
LIN {X 0,Y 390.318,Z 346.864,A -85,B 0,C 180,E1 -11793.096,E2 -11793.096} C_VEL
LIN {X 0,Y 390.327,Z 346.861,A -85,B 0,C 180,E1 -11796.202,E2 -11796.202} C_VEL
LIN {X 0,Y 390.207,Z 346.881,A -85,B 0,C 180,E1 -11799.328,E2 -11799.328} C_VEL
LIN {X 0,Y 390.173,Z 346.88,A -85,B 0,C 180,E1 -11802.483,E2 -11802.483} C_VEL
LIN {X 0,Y 390.141,Z 346.886,A -85,B 0,C 180,E1 -11805.676,E2 -11805.676} C_VEL
LIN {X 0,Y 390.107,Z 346.891,A -85,B 0,C 180,E1 -11808.921,E2 -11808.921} C_VEL
LIN {X 0,Y 390.04,Z 346.896,A -85,B 0,C 180,E1 -11812.233,E2 -11812.233} C_VEL
LIN {X 0,Y 390.119,Z 346.888,A -85,B 0,C 180,E1 -11815.743,E2 -11815.743} C_VEL
LIN {X 0,Y 390.058,Z 346.901,A -85,B 0,C 180,E1 -11819.109,E2 -11819.109} C_VEL
LIN {X 0,Y 390.01,Z 346.898,A -85,B 0,C 180,E1 -11820.823,E2 -11820.823} C_VEL
LIN {X 0,Y 389.337,Z 346.987,A -85,B 0,C 180,E1 -11821.685,E2 -11821.685} C_VEL
LIN {X 0,Y 386.489,Z 347.345,A -85,B 0,C 180,E1 -11823.087,E2 -11823.087} C_VEL
LIN {X 0,Y 384.091,Z 347.64,A -85,B 0,C 180,E1 -11824.219,E2 -11824.219} C_VEL
LIN {X 0,Y 383.074,Z 347.77,A -85,B 0,C 180,E1 -11825.095,E2 -11825.095} C_VEL
LIN {X 0,Y 382.997,Z 347.772,A -85,B 0,C 180,E1 -11825.392,E2 -11825.392} C_VEL
LIN {X 0,Y 383.006,Z 347.775,A -85,B 0,C 180,E1 -11828.599,E2 -11828.599} C_VEL
LIN {X 0,Y 383.043,Z 347.773,A -85,B 0,C 180,E1 -11831.338,E2 -11831.338} C_VEL
LIN {X 0,Y 383.124,Z 347.974,A -85,B 0,C 180,E1 -11834.582,E2 -11834.582} C_VEL
LIN {X 0,Y 383.289,Z 348.898,A -85,B 0,C 180,E1 -11834.738,E2 -11834.738} C_VEL
LIN {X 0,Y 386.601,Z 360.469,A -85,B 0,C 180,E1 -11835.682,E2 -11835.682} C_VEL
LIN {X 0,Y 387.68,Z 364.95,A -85,B 0,C 180,E1 -11836.092,E2 -11836.092} C_VEL
LIN {X 0,Y 386.912,Z 377.24,A -85,B 0,C 180,E1 -11837.243,E2 -11837.243} C_VEL
LIN {X 0,Y 386.264,Z 387.707,A -85,B 0,C 180,E1 -11838.473,E2 -11838.473} C_VEL
LIN {X 0,Y 385.498,Z 397.189,A -85,B 0,C 180,E1 -11839.85,E2 -11839.85} C_VEL
LIN {X 0,Y 384.839,Z 405.269,A -85,B 0,C 180,E1 -11841.282,E2 -11841.282} C_VEL
LIN {X 0,Y 384.309,Z 412.588,A -85,B 0,C 180,E1 -11842.88,E2 -11842.88} C_VEL
LIN {X 0,Y 383.834,Z 418.35,A -85,B 0,C 180,E1 -11844.455,E2 -11844.455} C_VEL
LIN {X 0,Y 383.472,Z 423.053,A -85,B 0,C 180,E1 -11846.088,E2 -11846.088} C_VEL
LIN {X 0,Y 383.206,Z 426.881,A -85,B 0,C 180,E1 -11847.869,E2 -11847.869} C_VEL
LIN {X 0,Y 383.05,Z 429.391,A -85,B 0,C 180,E1 -11849.577,E2 -11849.577} C_VEL
LIN {X 0,Y 382.999,Z 431.022,A -85,B 0,C 180,E1 -11851.736,E2 -11851.736} C_VEL
LIN {X 0,Y 383.126,Z 430.992,A -85,B 0,C 180,E1 -11853.88,E2 -11853.88} C_VEL
LIN {X 0,Y 383.298,Z 430.249,A -85,B 0,C 180,E1 -11855.057,E2 -11855.057} C_VEL
LIN {X 0,Y 383.55,Z 428.851,A -85,B 0,C 180,E1 -11856.37,E2 -11856.37} C_VEL
LIN {X 0,Y 383.951,Z 426.261,A -85,B 0,C 180,E1 -11857.961,E2 -11857.961} C_VEL
LIN {X 0,Y 384.451,Z 422.335,A -85,B 0,C 180,E1 -11859.676,E2 -11859.676} C_VEL
LIN {X 0,Y 385.246,Z 416.455,A -85,B 0,C 180,E1 -11861.551,E2 -11861.551} C_VEL
LIN {X 0,Y 385.965,Z 410.407,A -85,B 0,C 180,E1 -11863.062,E2 -11863.062} C_VEL
LIN {X 0,Y 386.869,Z 402.801,A -85,B 0,C 180,E1 -11864.588,E2 -11864.588} C_VEL
LIN {X 0,Y 387.652,Z 395.207,A -85,B 0,C 180,E1 -11865.833,E2 -11865.833} C_VEL
LIN {X 0,Y 388.588,Z 385.889,A -85,B 0,C 180,E1 -11867.081,E2 -11867.081} C_VEL
LIN {X 0,Y 389.481,Z 374.788,A -85,B 0,C 180,E1 -11868.286,E2 -11868.286} C_VEL
LIN {X 0,Y 389.699,Z 367.495,A -85,B 0,C 180,E1 -11868.953,E2 -11868.953} C_VEL
LIN {X 0,Y 386.711,Z 357.785,A -85,B 0,C 180,E1 -11869.926,E2 -11869.926} C_VEL
LIN {X 0,Y 383.312,Z 348.553,A -85,B 0,C 180,E1 -11870.768,E2 -11870.768} C_VEL
LIN {X 0,Y 383.166,Z 347.788,A -85,B 0,C 180,E1 -11871.031,E2 -11871.031} C_VEL
LIN {X 0,Y 383.271,Z 347.743,A -85,B 0,C 180,E1 -11873.683,E2 -11873.683} C_VEL
LIN {X 0,Y 383.375,Z 347.731,A -85,B 0,C 180,E1 -11877.899,E2 -11877.899} C_VEL
LIN {X 0,Y 383.509,Z 347.714,A -85,B 0,C 180,E1 -11880,E2 -11880} C_VEL
LIN {X 0,Y 383.235,Z 347.75,A -85,B 0,C 180,E1 -11883.154,E2 -11883.154} C_VEL
LIN {X 0,Y 383.261,Z 347.743,A -85,B 0,C 180,E1 -11886.317,E2 -11886.317} C_VEL
LIN {X 0,Y 383.134,Z 347.76,A -85,B 0,C 180,E1 -11889.503,E2 -11889.503} C_VEL
LIN {X 0,Y 383.117,Z 347.762,A -85,B 0,C 180,E1 -11893.536,E2 -11893.536} C_VEL
LIN {X 0,Y 383.085,Z 347.763,A -85,B 0,C 180,E1 -11897.07,E2 -11897.07} C_VEL
LIN {X 0,Y 383.02,Z 347.77,A -85,B 0,C 180,E1 -11900.647,E2 -11900.647} C_VEL
LIN {X 0,Y 383.015,Z 347.77,A -85,B 0,C 180,E1 -11903.809,E2 -11903.809} C_VEL
LIN {X 0,Y 383.072,Z 347.764,A -85,B 0,C 180,E1 -11906.124,E2 -11906.124} C_VEL
LIN {X 0,Y 382.985,Z 347.779,A -85,B 0,C 180,E1 -11909.701,E2 -11909.701} C_VEL
LIN {X 0,Y 382.996,Z 347.776,A -85,B 0,C 180,E1 -11913.402,E2 -11913.402} C_VEL
LIN {X 0,Y 383.025,Z 347.775,A -85,B 0,C 180,E1 -11916.165,E2 -11916.165} C_VEL
LIN {X 0,Y 382.969,Z 347.781,A -85,B 0,C 180,E1 -11919.964,E2 -11919.964} C_VEL
LIN {X 0,Y 383.001,Z 347.778,A -85,B 0,C 180,E1 -11922.779,E2 -11922.779} C_VEL
LIN {X 0,Y 383.032,Z 347.968,A -85,B 0,C 180,E1 -11925.132,E2 -11925.132} C_VEL
LIN {X 0,Y 384.559,Z 355.458,A -85,B 0,C 180,E1 -11928.53,E2 -11928.53} C_VEL
LIN {X 0,Y 386.1,Z 363.496,A -85,B 0,C 180,E1 -11931.766,E2 -11931.766} C_VEL
LIN {X 0,Y 386.441,Z 367.245,A -85,B 0,C 180,E1 -11933.15,E2 -11933.15} C_VEL
LIN {X 0,Y 384.926,Z 380.592,A -85,B 0,C 180,E1 -11937.556,E2 -11937.556} C_VEL
LIN {X 0,Y 384.08,Z 391.609,A -85,B 0,C 180,E1 -11940.995,E2 -11940.995} C_VEL
LIN {X 0,Y 383.323,Z 403.247,A -85,B 0,C 180,E1 -11944.479,E2 -11944.479} C_VEL
LIN {X 0,Y 382.78,Z 415.005,A -85,B 0,C 180,E1 -11947.89,E2 -11947.89} C_VEL
LIN {X 0,Y 382.535,Z 424.091,A -85,B 0,C 180,E1 -11950.41,E2 -11950.41} C_VEL
LIN {X 0,Y 382.966,Z 427.106,A -85,B 0,C 180,E1 -11950.58,E2 -11950.58} C_VEL
LIN {X 0,Y 384.752,Z 440.291,A -85,B 0,C 180,E1 -11951.17,E2 -11951.17} C_VEL
LIN {X 0,Y 385.675,Z 453.096,A -85,B 0,C 180,E1 -11951.891,E2 -11951.891} C_VEL
LIN {X 0,Y 385.847,Z 465.771,A -85,B 0,C 180,E1 -11952.784,E2 -11952.784} C_VEL
LIN {X 0,Y 385.877,Z 475.297,A -85,B 0,C 180,E1 -11953.603,E2 -11953.603} C_VEL
LIN {X 0,Y 384.69,Z 486.912,A -85,B 0,C 180,E1 -11954.775,E2 -11954.775} C_VEL
LIN {X 0,Y 383.735,Z 497.493,A -85,B 0,C 180,E1 -11956.092,E2 -11956.092} C_VEL
LIN {X 0,Y 383.215,Z 505.41,A -85,B 0,C 180,E1 -11957.287,E2 -11957.287} C_VEL
LIN {X 0,Y 382.585,Z 514.15,A -85,B 0,C 180,E1 -11958.879,E2 -11958.879} C_VEL
LIN {X 0,Y 382.229,Z 521.287,A -85,B 0,C 180,E1 -11960.475,E2 -11960.475} C_VEL
LIN {X 0,Y 382.152,Z 527.075,A -85,B 0,C 180,E1 -11962.072,E2 -11962.072} C_VEL
LIN {X 0,Y 382.215,Z 531.658,A -85,B 0,C 180,E1 -11963.666,E2 -11963.666} C_VEL
LIN {X 0,Y 382.261,Z 534.112,A -85,B 0,C 180,E1 -11964.726,E2 -11964.726} C_VEL
LIN {X 0,Y 382.447,Z 536.078,A -85,B 0,C 180,E1 -11965.785,E2 -11965.785} C_VEL
LIN {X 0,Y 382.456,Z 537.59,A -85,B 0,C 180,E1 -11966.84,E2 -11966.84} C_VEL
LIN {X 0,Y 382.493,Z 538.689,A -85,B 0,C 180,E1 -11967.894,E2 -11967.894} C_VEL
LIN {X 0,Y 382.777,Z 539.373,A -85,B 0,C 180,E1 -11968.948,E2 -11968.948} C_VEL
LIN {X 0,Y 382.811,Z 539.578,A -85,B 0,C 180,E1 -11970,E2 -11970} C_VEL
LIN {X 0,Y 382.772,Z 539.365,A -85,B 0,C 180,E1 -11971.052,E2 -11971.052} C_VEL
LIN {X 0,Y 382.497,Z 538.706,A -85,B 0,C 180,E1 -11972.106,E2 -11972.106} C_VEL
LIN {X 0,Y 382.461,Z 537.609,A -85,B 0,C 180,E1 -11973.16,E2 -11973.16} C_VEL
LIN {X 0,Y 382.483,Z 536.08,A -85,B 0,C 180,E1 -11974.215,E2 -11974.215} C_VEL
LIN {X 0,Y 382.273,Z 532.887,A -85,B 0,C 180,E1 -11975.803,E2 -11975.803} C_VEL
LIN {X 0,Y 382.191,Z 528.585,A -85,B 0,C 180,E1 -11977.396,E2 -11977.396} C_VEL
LIN {X 0,Y 382.196,Z 523.054,A -85,B 0,C 180,E1 -11978.992,E2 -11978.992} C_VEL
LIN {X 0,Y 382.413,Z 516.137,A -85,B 0,C 180,E1 -11980.59,E2 -11980.59} C_VEL
LIN {X 0,Y 382.836,Z 509.089,A -85,B 0,C 180,E1 -11981.918,E2 -11981.918} C_VEL
LIN {X 0,Y 383.453,Z 500.599,A -85,B 0,C 180,E1 -11983.244,E2 -11983.244} C_VEL
LIN {X 0,Y 384.184,Z 490.409,A -85,B 0,C 180,E1 -11984.541,E2 -11984.541} C_VEL
LIN {X 0,Y 384.997,Z 479.977,A -85,B 0,C 180,E1 -11985.62,E2 -11985.62} C_VEL
LIN {X 0,Y 385.575,Z 472.327,A -85,B 0,C 180,E1 -11986.274,E2 -11986.274} C_VEL
LIN {X 0,Y 384.954,Z 459.115,A -85,B 0,C 180,E1 -11987.227,E2 -11987.227} C_VEL
LIN {X 0,Y 384.017,Z 446.361,A -85,B 0,C 180,E1 -11987.927,E2 -11987.927} C_VEL
LIN {X 0,Y 382.731,Z 433.039,A -85,B 0,C 180,E1 -11988.449,E2 -11988.449} C_VEL
LIN {X 0,Y 382.473,Z 430.19,A -85,B 0,C 180,E1 -11988.583,E2 -11988.583} C_VEL
LIN {X 0,Y 382.97,Z 417.949,A -85,B 0,C 180,E1 -11992.098,E2 -11992.098} C_VEL
LIN {X 0,Y 383.622,Z 406.415,A -85,B 0,C 180,E1 -11995.5,E2 -11995.5} C_VEL
LIN {X 0,Y 384.401,Z 394.571,A -85,B 0,C 180,E1 -11999.046,E2 -11999.046} C_VEL
LIN {X 0,Y 385.216,Z 385.063,A -85,B 0,C 180,E1 -12001.943,E2 -12001.943} C_VEL
LIN {X 0,Y 386.379,Z 373.325,A -85,B 0,C 180,E1 -12005.595,E2 -12005.595} C_VEL
LIN {X 0,Y 386.881,Z 369.083,A -85,B 0,C 180,E1 -12006.937,E2 -12006.937} C_VEL
LIN {X 0,Y 386.272,Z 364.394,A -85,B 0,C 180,E1 -12008.522,E2 -12008.522} C_VEL
LIN {X 0,Y 384.614,Z 356.018,A -85,B 0,C 180,E1 -12011.48,E2 -12011.48} C_VEL
LIN {X 0,Y 383.025,Z 347.853,A -85,B 0,C 180,E1 -12014.547,E2 -12014.547} C_VEL
LIN {X 0,Y 383.006,Z 347.778,A -85,B 0,C 180,E1 -12017.239,E2 -12017.239} C_VEL
LIN {X 0,Y 382.98,Z 347.776,A -85,B 0,C 180,E1 -12020.418,E2 -12020.418} C_VEL
LIN {X 0,Y 383.018,Z 347.771,A -85,B 0,C 180,E1 -12024.043,E2 -12024.043} C_VEL
LIN {X 0,Y 382.979,Z 347.779,A -85,B 0,C 180,E1 -12027.578,E2 -12027.578} C_VEL
LIN {X 0,Y 382.985,Z 347.775,A -85,B 0,C 180,E1 -12030.299,E2 -12030.299} C_VEL
LIN {X 0,Y 383.073,Z 347.764,A -85,B 0,C 180,E1 -12034.02,E2 -12034.02} C_VEL
LIN {X 0,Y 382.983,Z 347.78,A -85,B 0,C 180,E1 -12037.334,E2 -12037.334} C_VEL
LIN {X 0,Y 383.05,Z 347.77,A -85,B 0,C 180,E1 -12040.716,E2 -12040.716} C_VEL
LIN {X 0,Y 383.071,Z 347.764,A -85,B 0,C 180,E1 -12044.026,E2 -12044.026} C_VEL
LIN {X 0,Y 383.127,Z 347.761,A -85,B 0,C 180,E1 -12047.284,E2 -12047.284} C_VEL
LIN {X 0,Y 383.134,Z 347.759,A -85,B 0,C 180,E1 -12050.497,E2 -12050.497} C_VEL
LIN {X 0,Y 383.261,Z 347.741,A -85,B 0,C 180,E1 -12053.683,E2 -12053.683} C_VEL
LIN {X 0,Y 383.375,Z 347.726,A -85,B 0,C 180,E1 -12057.899,E2 -12057.899} C_VEL
LIN {X 0,Y 383.509,Z 347.71,A -85,B 0,C 180,E1 -12060,E2 -12060} C_VEL
LIN {X 0,Y 383.234,Z 347.746,A -85,B 0,C 180,E1 -12063.154,E2 -12063.154} C_VEL
LIN {X 0,Y 383.248,Z 347.742,A -85,B 0,C 180,E1 -12066.697,E2 -12066.697} C_VEL
LIN {X 0,Y 383.142,Z 347.755,A -85,B 0,C 180,E1 -12069.502,E2 -12069.502} C_VEL
LIN {X 0,Y 383.117,Z 347.759,A -85,B 0,C 180,E1 -12073.536,E2 -12073.536} C_VEL
LIN {X 0,Y 383.086,Z 347.762,A -85,B 0,C 180,E1 -12077.455,E2 -12077.455} C_VEL
LIN {X 0,Y 383.027,Z 347.775,A -85,B 0,C 180,E1 -12080.65,E2 -12080.65} C_VEL
LIN {X 0,Y 383.026,Z 347.771,A -85,B 0,C 180,E1 -12083.808,E2 -12083.808} C_VEL
LIN {X 0,Y 383.05,Z 347.767,A -85,B 0,C 180,E1 -12087.302,E2 -12087.302} C_VEL
LIN {X 0,Y 382.979,Z 347.777,A -85,B 0,C 180,E1 -12090.919,E2 -12090.919} C_VEL
LIN {X 0,Y 383.012,Z 347.775,A -85,B 0,C 180,E1 -12094.669,E2 -12094.669} C_VEL
LIN {X 0,Y 382.997,Z 347.776,A -85,B 0,C 180,E1 -12097.905,E2 -12097.905} C_VEL
LIN {X 0,Y 383.008,Z 347.772,A -85,B 0,C 180,E1 -12101.344,E2 -12101.344} C_VEL
LIN {X 0,Y 382.993,Z 347.779,A -85,B 0,C 180,E1 -12104.304,E2 -12104.304} C_VEL
LIN {X 0,Y 383.006,Z 347.772,A -85,B 0,C 180,E1 -12107.241,E2 -12107.241} C_VEL
LIN {X 0,Y 383.014,Z 347.775,A -85,B 0,C 180,E1 -12110.414,E2 -12110.414} C_VEL
LIN {X 0,Y 383.024,Z 347.777,A -85,B 0,C 180,E1 -12114.045,E2 -12114.045} C_VEL
LIN {X 0,Y 383.035,Z 347.774,A -85,B 0,C 180,E1 -12117.854,E2 -12117.854} C_VEL
LIN {X 0,Y 383.063,Z 347.77,A -85,B 0,C 180,E1 -12121.721,E2 -12121.721} C_VEL
LIN {X 0,Y 383.052,Z 347.767,A -85,B 0,C 180,E1 -12125.04,E2 -12125.04} C_VEL
LIN {X 0,Y 382.994,Z 347.775,A -85,B 0,C 180,E1 -12128.47,E2 -12128.47} C_VEL
LIN {X 0,Y 383.091,Z 347.768,A -85,B 0,C 180,E1 -12131.828,E2 -12131.828} C_VEL
LIN {X 0,Y 383.115,Z 347.76,A -85,B 0,C 180,E1 -12135.119,E2 -12135.119} C_VEL
LIN {X 0,Y 383.1,Z 347.761,A -85,B 0,C 180,E1 -12138.358,E2 -12138.358} C_VEL
LIN {X 0,Y 383.306,Z 347.739,A -85,B 0,C 180,E1 -12141.933,E2 -12141.933} C_VEL
LIN {X 0,Y 383.203,Z 347.748,A -85,B 0,C 180,E1 -12144.739,E2 -12144.739} C_VEL
LIN {X 0,Y 383.39,Z 347.728,A -85,B 0,C 180,E1 -12147.899,E2 -12147.899} C_VEL
LIN {X 0,Y 383.522,Z 347.71,A -85,B 0,C 180,E1 -12150,E2 -12150} C_VEL
LIN {X 0,Y 383.255,Z 347.744,A -85,B 0,C 180,E1 -12153.154,E2 -12153.154} C_VEL
LIN {X 0,Y 383.283,Z 347.738,A -85,B 0,C 180,E1 -12156.316,E2 -12156.316} C_VEL
LIN {X 0,Y 383.154,Z 347.76,A -85,B 0,C 180,E1 -12159.502,E2 -12159.502} C_VEL
LIN {X 0,Y 383.127,Z 347.762,A -85,B 0,C 180,E1 -12163.536,E2 -12163.536} C_VEL
LIN {X 0,Y 383.096,Z 347.766,A -85,B 0,C 180,E1 -12167.454,E2 -12167.454} C_VEL
LIN {X 0,Y 383.029,Z 347.77,A -85,B 0,C 180,E1 -12170.646,E2 -12170.646} C_VEL
LIN {X 0,Y 383.033,Z 347.77,A -85,B 0,C 180,E1 -12173.807,E2 -12173.807} C_VEL
LIN {X 0,Y 383.08,Z 347.763,A -85,B 0,C 180,E1 -12176.123,E2 -12176.123} C_VEL
LIN {X 0,Y 382.991,Z 347.775,A -85,B 0,C 180,E1 -12179.699,E2 -12179.699} C_VEL
LIN {X 0,Y 383.001,Z 347.776,A -85,B 0,C 180,E1 -12183.4,E2 -12183.4} C_VEL
LIN {X 0,Y 382.997,Z 347.772,A -85,B 0,C 180,E1 -12185.392,E2 -12185.392} C_VEL
LIN {X 0,Y 382.355,Z 347.854,A -85,B 0,C 180,E1 -12186.27,E2 -12186.27} C_VEL
LIN {X 0,Y 379.538,Z 348.207,A -85,B 0,C 180,E1 -12187.698,E2 -12187.698} C_VEL
LIN {X 0,Y 377.132,Z 348.509,A -85,B 0,C 180,E1 -12188.852,E2 -12188.852} C_VEL
LIN {X 0,Y 376.085,Z 348.638,A -85,B 0,C 180,E1 -12189.744,E2 -12189.744} C_VEL
LIN {X 0,Y 375.993,Z 348.649,A -85,B 0,C 180,E1 -12190.046,E2 -12190.046} C_VEL
LIN {X 0,Y 375.999,Z 348.649,A -85,B 0,C 180,E1 -12193.754,E2 -12193.754} C_VEL
LIN {X 0,Y 376.082,Z 348.934,A -85,B 0,C 180,E1 -12194.327,E2 -12194.327} C_VEL
LIN {X 0,Y 376.449,Z 350.314,A -85,B 0,C 180,E1 -12194.508,E2 -12194.508} C_VEL
LIN {X 0,Y 379.903,Z 362.629,A -85,B 0,C 180,E1 -12195.547,E2 -12195.547} C_VEL
LIN {X 0,Y 380.779,Z 366.593,A -85,B 0,C 180,E1 -12195.92,E2 -12195.92} C_VEL
LIN {X 0,Y 380.003,Z 378.822,A -85,B 0,C 180,E1 -12197.098,E2 -12197.098} C_VEL
LIN {X 0,Y 379.311,Z 389.08,A -85,B 0,C 180,E1 -12198.34,E2 -12198.34} C_VEL
LIN {X 0,Y 378.467,Z 399.152,A -85,B 0,C 180,E1 -12199.848,E2 -12199.848} C_VEL
LIN {X 0,Y 377.797,Z 407.424,A -85,B 0,C 180,E1 -12201.379,E2 -12201.379} C_VEL
LIN {X 0,Y 377.262,Z 414.58,A -85,B 0,C 180,E1 -12203.034,E2 -12203.034} C_VEL
LIN {X 0,Y 376.743,Z 420.259,A -85,B 0,C 180,E1 -12204.669,E2 -12204.669} C_VEL
LIN {X 0,Y 376.394,Z 425.357,A -85,B 0,C 180,E1 -12206.577,E2 -12206.577} C_VEL
LIN {X 0,Y 376.117,Z 428.896,A -85,B 0,C 180,E1 -12208.453,E2 -12208.453} C_VEL
LIN {X 0,Y 376.013,Z 430.534,A -85,B 0,C 180,E1 -12209.692,E2 -12209.692} C_VEL
LIN {X 0,Y 375.966,Z 431.936,A -85,B 0,C 180,E1 -12211.469,E2 -12211.469} C_VEL
LIN {X 0,Y 376.09,Z 432.095,A -85,B 0,C 180,E1 -12213.76,E2 -12213.76} C_VEL
LIN {X 0,Y 376.424,Z 430.792,A -85,B 0,C 180,E1 -12215.748,E2 -12215.748} C_VEL
LIN {X 0,Y 376.689,Z 429.31,A -85,B 0,C 180,E1 -12216.933,E2 -12216.933} C_VEL
LIN {X 0,Y 377.211,Z 426.205,A -85,B 0,C 180,E1 -12218.678,E2 -12218.678} C_VEL
LIN {X 0,Y 377.773,Z 421.863,A -85,B 0,C 180,E1 -12220.435,E2 -12220.435} C_VEL
LIN {X 0,Y 378.545,Z 416.206,A -85,B 0,C 180,E1 -12222.161,E2 -12222.161} C_VEL
LIN {X 0,Y 379.504,Z 408.965,A -85,B 0,C 180,E1 -12223.872,E2 -12223.872} C_VEL
LIN {X 0,Y 380.356,Z 401.581,A -85,B 0,C 180,E1 -12225.282,E2 -12225.282} C_VEL
LIN {X 0,Y 381.362,Z 392.606,A -85,B 0,C 180,E1 -12226.682,E2 -12226.682} C_VEL
LIN {X 0,Y 382.405,Z 381.977,A -85,B 0,C 180,E1 -12228.005,E2 -12228.005} C_VEL
LIN {X 0,Y 383.296,Z 370.532,A -85,B 0,C 180,E1 -12229.145,E2 -12229.145} C_VEL
LIN {X 0,Y 381.288,Z 363.225,A -85,B 0,C 180,E1 -12229.916,E2 -12229.916} C_VEL
LIN {X 0,Y 377.652,Z 353.081,A -85,B 0,C 180,E1 -12230.899,E2 -12230.899} C_VEL
LIN {X 0,Y 376.252,Z 349.309,A -85,B 0,C 180,E1 -12231.271,E2 -12231.271} C_VEL
LIN {X 0,Y 376.188,Z 348.655,A -85,B 0,C 180,E1 -12231.519,E2 -12231.519} C_VEL
LIN {X 0,Y 376.158,Z 348.629,A -85,B 0,C 180,E1 -12234.64,E2 -12234.64} C_VEL
LIN {X 0,Y 376.341,Z 348.608,A -85,B 0,C 180,E1 -12237.86,E2 -12237.86} C_VEL
LIN {X 0,Y 376.479,Z 348.59,A -85,B 0,C 180,E1 -12240,E2 -12240} C_VEL
LIN {X 0,Y 376.173,Z 348.629,A -85,B 0,C 180,E1 -12243.213,E2 -12243.213} C_VEL
LIN {X 0,Y 376.218,Z 348.621,A -85,B 0,C 180,E1 -12246.436,E2 -12246.436} C_VEL
LIN {X 0,Y 376.104,Z 348.634,A -85,B 0,C 180,E1 -12249.682,E2 -12249.682} C_VEL
LIN {X 0,Y 376.081,Z 348.638,A -85,B 0,C 180,E1 -12253.658,E2 -12253.658} C_VEL
LIN {X 0,Y 376.024,Z 348.64,A -85,B 0,C 180,E1 -12257.4,E2 -12257.4} C_VEL
LIN {X 0,Y 375.971,Z 348.648,A -85,B 0,C 180,E1 -12260.833,E2 -12260.833} C_VEL
LIN {X 0,Y 375.98,Z 348.648,A -85,B 0,C 180,E1 -12264.283,E2 -12264.283} C_VEL
LIN {X 0,Y 376.013,Z 348.644,A -85,B 0,C 180,E1 -12266.653,E2 -12266.653} C_VEL
LIN {X 0,Y 375.958,Z 348.655,A -85,B 0,C 180,E1 -12270.313,E2 -12270.313} C_VEL
LIN {X 0,Y 375.954,Z 348.654,A -85,B 0,C 180,E1 -12274.112,E2 -12274.112} C_VEL
LIN {X 0,Y 375.946,Z 348.656,A -85,B 0,C 180,E1 -12276.742,E2 -12276.742} C_VEL
LIN {X 0,Y 375.933,Z 348.658,A -85,B 0,C 180,E1 -12279.962,E2 -12279.962} C_VEL
LIN {X 0,Y 375.92,Z 348.658,A -85,B 0,C 180,E1 -12283.768,E2 -12283.768} C_VEL
LIN {X 0,Y 375.98,Z 348.774,A -85,B 0,C 180,E1 -12284.512,E2 -12284.512} C_VEL
LIN {X 0,Y 377.147,Z 354.528,A -85,B 0,C 180,E1 -12287.281,E2 -12287.281} C_VEL
LIN {X 0,Y 378.515,Z 361.452,A -85,B 0,C 180,E1 -12290.262,E2 -12290.262} C_VEL
LIN {X 0,Y 379.454,Z 366.648,A -85,B 0,C 180,E1 -12292.325,E2 -12292.325} C_VEL
LIN {X 0,Y 379.235,Z 370.268,A -85,B 0,C 180,E1 -12293.629,E2 -12293.629} C_VEL
LIN {X 0,Y 377.963,Z 381.39,A -85,B 0,C 180,E1 -12297.369,E2 -12297.369} C_VEL
LIN {X 0,Y 377.027,Z 392.788,A -85,B 0,C 180,E1 -12301.011,E2 -12301.011} C_VEL
LIN {X 0,Y 376.235,Z 404.385,A -85,B 0,C 180,E1 -12304.556,E2 -12304.556} C_VEL
LIN {X 0,Y 375.68,Z 416.091,A -85,B 0,C 180,E1 -12308.029,E2 -12308.029} C_VEL
LIN {X 0,Y 375.507,Z 422.679,A -85,B 0,C 180,E1 -12309.906,E2 -12309.906} C_VEL
LIN {X 0,Y 375.761,Z 424.964,A -85,B 0,C 180,E1 -12310.065,E2 -12310.065} C_VEL
LIN {X 0,Y 377.868,Z 438.937,A -85,B 0,C 180,E1 -12310.726,E2 -12310.726} C_VEL
LIN {X 0,Y 378.819,Z 451.547,A -85,B 0,C 180,E1 -12311.457,E2 -12311.457} C_VEL
LIN {X 0,Y 378.964,Z 463.748,A -85,B 0,C 180,E1 -12312.322,E2 -12312.322} C_VEL
LIN {X 0,Y 378.898,Z 476.239,A -85,B 0,C 180,E1 -12313.431,E2 -12313.431} C_VEL
LIN {X 0,Y 377.679,Z 487.5,A -85,B 0,C 180,E1 -12314.623,E2 -12314.623} C_VEL
LIN {X 0,Y 376.704,Z 497.665,A -85,B 0,C 180,E1 -12315.964,E2 -12315.964} C_VEL
LIN {X 0,Y 376.268,Z 504.603,A -85,B 0,C 180,E1 -12317.048,E2 -12317.048} C_VEL
LIN {X 0,Y 375.575,Z 513.285,A -85,B 0,C 180,E1 -12318.669,E2 -12318.669} C_VEL
LIN {X 0,Y 375.156,Z 520.392,A -85,B 0,C 180,E1 -12320.294,E2 -12320.294} C_VEL
LIN {X 0,Y 375.078,Z 526.158,A -85,B 0,C 180,E1 -12321.922,E2 -12321.922} C_VEL
LIN {X 0,Y 375.135,Z 530.717,A -85,B 0,C 180,E1 -12323.546,E2 -12323.546} C_VEL
LIN {X 0,Y 375.185,Z 533.148,A -85,B 0,C 180,E1 -12324.626,E2 -12324.626} C_VEL
LIN {X 0,Y 375.37,Z 535.1,A -85,B 0,C 180,E1 -12325.705,E2 -12325.705} C_VEL
LIN {X 0,Y 375.406,Z 536.606,A -85,B 0,C 180,E1 -12326.78,E2 -12326.78} C_VEL
LIN {X 0,Y 375.45,Z 537.698,A -85,B 0,C 180,E1 -12327.855,E2 -12327.855} C_VEL
LIN {X 0,Y 375.747,Z 538.361,A -85,B 0,C 180,E1 -12328.928,E2 -12328.928} C_VEL
LIN {X 0,Y 375.786,Z 538.562,A -85,B 0,C 180,E1 -12330,E2 -12330} C_VEL
LIN {X 0,Y 375.742,Z 538.34,A -85,B 0,C 180,E1 -12331.072,E2 -12331.072} C_VEL
LIN {X 0,Y 375.461,Z 537.665,A -85,B 0,C 180,E1 -12332.145,E2 -12332.145} C_VEL
LIN {X 0,Y 375.423,Z 536.549,A -85,B 0,C 180,E1 -12333.219,E2 -12333.219} C_VEL
LIN {X 0,Y 375.333,Z 534.057,A -85,B 0,C 180,E1 -12334.833,E2 -12334.833} C_VEL
LIN {X 0,Y 375.167,Z 529.416,A -85,B 0,C 180,E1 -12336.855,E2 -12336.855} C_VEL
LIN {X 0,Y 375.115,Z 523.903,A -85,B 0,C 180,E1 -12338.62,E2 -12338.62} C_VEL
LIN {X 0,Y 375.276,Z 517.395,A -85,B 0,C 180,E1 -12340.248,E2 -12340.248} C_VEL
LIN {X 0,Y 375.737,Z 509.309,A -85,B 0,C 180,E1 -12341.873,E2 -12341.873} C_VEL
LIN {X 0,Y 376.364,Z 501.285,A -85,B 0,C 180,E1 -12343.193,E2 -12343.193} C_VEL
LIN {X 0,Y 377.085,Z 491.511,A -85,B 0,C 180,E1 -12344.517,E2 -12344.517} C_VEL
LIN {X 0,Y 377.897,Z 481.216,A -85,B 0,C 180,E1 -12345.644,E2 -12345.644} C_VEL
LIN {X 0,Y 378.511,Z 472.345,A -85,B 0,C 180,E1 -12346.448,E2 -12346.448} C_VEL
LIN {X 0,Y 377.992,Z 459.961,A -85,B 0,C 180,E1 -12347.376,E2 -12347.376} C_VEL
LIN {X 0,Y 377.076,Z 446.947,A -85,B 0,C 180,E1 -12348.135,E2 -12348.135} C_VEL
LIN {X 0,Y 375.706,Z 432.45,A -85,B 0,C 180,E1 -12348.736,E2 -12348.736} C_VEL
LIN {X 0,Y 375.429,Z 429.383,A -85,B 0,C 180,E1 -12348.874,E2 -12348.874} C_VEL
LIN {X 0,Y 375.97,Z 416.891,A -85,B 0,C 180,E1 -12352.532,E2 -12352.532} C_VEL
LIN {X 0,Y 376.732,Z 403.955,A -85,B 0,C 180,E1 -12356.434,E2 -12356.434} C_VEL
LIN {X 0,Y 377.664,Z 391.847,A -85,B 0,C 180,E1 -12360.161,E2 -12360.161} C_VEL
LIN {X 0,Y 378.75,Z 380.147,A -85,B 0,C 180,E1 -12363.825,E2 -12363.825} C_VEL
LIN {X 0,Y 379.844,Z 370.894,A -85,B 0,C 180,E1 -12366.797,E2 -12366.797} C_VEL
LIN {X 0,Y 379.467,Z 366.624,A -85,B 0,C 180,E1 -12368.249,E2 -12368.249} C_VEL
LIN {X 0,Y 377.852,Z 358.328,A -85,B 0,C 180,E1 -12371.22,E2 -12371.22} C_VEL
LIN {X 0,Y 375.999,Z 348.735,A -85,B 0,C 180,E1 -12374.858,E2 -12374.858} C_VEL
LIN {X 0,Y 375.912,Z 348.657,A -85,B 0,C 180,E1 -12378.402,E2 -12378.402} C_VEL
LIN {X 0,Y 375.948,Z 348.653,A -85,B 0,C 180,E1 -12381.909,E2 -12381.909} C_VEL
LIN {X 0,Y 375.974,Z 348.655,A -85,B 0,C 180,E1 -12385.332,E2 -12385.332} C_VEL
LIN {X 0,Y 375.95,Z 348.651,A -85,B 0,C 180,E1 -12388.437,E2 -12388.437} C_VEL
LIN {X 0,Y 375.976,Z 348.648,A -85,B 0,C 180,E1 -12392.14,E2 -12392.14} C_VEL
LIN {X 0,Y 375.998,Z 348.646,A -85,B 0,C 180,E1 -12394.538,E2 -12394.538} C_VEL
LIN {X 0,Y 375.948,Z 348.652,A -85,B 0,C 180,E1 -12398.045,E2 -12398.045} C_VEL
LIN {X 0,Y 375.994,Z 348.648,A -85,B 0,C 180,E1 -12401.472,E2 -12401.472} C_VEL
LIN {X 0,Y 376.049,Z 348.644,A -85,B 0,C 180,E1 -12404.832,E2 -12404.832} C_VEL
LIN {X 0,Y 376.04,Z 348.64,A -85,B 0,C 180,E1 -12408.136,E2 -12408.136} C_VEL
LIN {X 0,Y 376.19,Z 348.621,A -85,B 0,C 180,E1 -12411.94,E2 -12411.94} C_VEL
LIN {X 0,Y 376.155,Z 348.63,A -85,B 0,C 180,E1 -12414.64,E2 -12414.64} C_VEL
LIN {X 0,Y 376.341,Z 348.603,A -85,B 0,C 180,E1 -12417.86,E2 -12417.86} C_VEL
LIN {X 0,Y 376.479,Z 348.586,A -85,B 0,C 180,E1 -12420,E2 -12420} C_VEL
LIN {X 0,Y 376.173,Z 348.626,A -85,B 0,C 180,E1 -12423.213,E2 -12423.213} C_VEL
LIN {X 0,Y 376.212,Z 348.62,A -85,B 0,C 180,E1 -12426.687,E2 -12426.687} C_VEL
LIN {X 0,Y 376.11,Z 348.631,A -85,B 0,C 180,E1 -12429.682,E2 -12429.682} C_VEL
LIN {X 0,Y 376.081,Z 348.635,A -85,B 0,C 180,E1 -12433.658,E2 -12433.658} C_VEL
LIN {X 0,Y 376.036,Z 348.641,A -85,B 0,C 180,E1 -12437.608,E2 -12437.608} C_VEL
LIN {X 0,Y 375.971,Z 348.652,A -85,B 0,C 180,E1 -12440.833,E2 -12440.833} C_VEL
LIN {X 0,Y 375.987,Z 348.651,A -85,B 0,C 180,E1 -12444.282,E2 -12444.282} C_VEL
LIN {X 0,Y 376.013,Z 348.648,A -85,B 0,C 180,E1 -12446.653,E2 -12446.653} C_VEL
LIN {X 0,Y 375.969,Z 348.65,A -85,B 0,C 180,E1 -12449.079,E2 -12449.079} C_VEL
LIN {X 0,Y 375.943,Z 348.654,A -85,B 0,C 180,E1 -12452.829,E2 -12452.829} C_VEL
LIN {X 0,Y 375.952,Z 348.651,A -85,B 0,C 180,E1 -12455.416,E2 -12455.416} C_VEL
LIN {X 0,Y 375.972,Z 348.655,A -85,B 0,C 180,E1 -12458.272,E2 -12458.272} C_VEL
LIN {X 0,Y 375.955,Z 348.652,A -85,B 0,C 180,E1 -12461.606,E2 -12461.606} C_VEL
LIN {X 0,Y 375.925,Z 348.655,A -85,B 0,C 180,E1 -12465.269,E2 -12465.269} C_VEL
LIN {X 0,Y 375.938,Z 348.656,A -85,B 0,C 180,E1 -12468.399,E2 -12468.399} C_VEL
LIN {X 0,Y 375.973,Z 348.651,A -85,B 0,C 180,E1 -12471.73,E2 -12471.73} C_VEL
LIN {X 0,Y 375.978,Z 348.648,A -85,B 0,C 180,E1 -12475.333,E2 -12475.333} C_VEL
LIN {X 0,Y 375.975,Z 348.65,A -85,B 0,C 180,E1 -12478.441,E2 -12478.441} C_VEL
LIN {X 0,Y 376.002,Z 348.649,A -85,B 0,C 180,E1 -12482.143,E2 -12482.143} C_VEL
LIN {X 0,Y 376.006,Z 348.645,A -85,B 0,C 180,E1 -12484.54,E2 -12484.54} C_VEL
LIN {X 0,Y 375.964,Z 348.654,A -85,B 0,C 180,E1 -12488.046,E2 -12488.046} C_VEL
LIN {X 0,Y 376.025,Z 348.645,A -85,B 0,C 180,E1 -12491.475,E2 -12491.475} C_VEL
LIN {X 0,Y 376.063,Z 348.637,A -85,B 0,C 180,E1 -12494.833,E2 -12494.833} C_VEL
LIN {X 0,Y 376.052,Z 348.641,A -85,B 0,C 180,E1 -12498.137,E2 -12498.137} C_VEL
LIN {X 0,Y 376.26,Z 348.617,A -85,B 0,C 180,E1 -12501.877,E2 -12501.877} C_VEL
LIN {X 0,Y 376.175,Z 348.623,A -85,B 0,C 180,E1 -12504.64,E2 -12504.64} C_VEL
LIN {X 0,Y 376.356,Z 348.604,A -85,B 0,C 180,E1 -12507.86,E2 -12507.86} C_VEL
LIN {X 0,Y 376.492,Z 348.586,A -85,B 0,C 180,E1 -12510,E2 -12510} C_VEL
LIN {X 0,Y 376.193,Z 348.625,A -85,B 0,C 180,E1 -12513.213,E2 -12513.213} C_VEL
LIN {X 0,Y 376.241,Z 348.615,A -85,B 0,C 180,E1 -12516.435,E2 -12516.435} C_VEL
LIN {X 0,Y 376.121,Z 348.634,A -85,B 0,C 180,E1 -12519.681,E2 -12519.681} C_VEL
LIN {X 0,Y 376.091,Z 348.637,A -85,B 0,C 180,E1 -12523.657,E2 -12523.657} C_VEL
LIN {X 0,Y 376.044,Z 348.643,A -85,B 0,C 180,E1 -12527.607,E2 -12527.607} C_VEL
LIN {X 0,Y 375.978,Z 348.65,A -85,B 0,C 180,E1 -12530.832,E2 -12530.832} C_VEL
LIN {X 0,Y 375.994,Z 348.646,A -85,B 0,C 180,E1 -12534.281,E2 -12534.281} C_VEL
LIN {X 0,Y 376.019,Z 348.644,A -85,B 0,C 180,E1 -12536.651,E2 -12536.651} C_VEL
LIN {X 0,Y 375.963,Z 348.65,A -85,B 0,C 180,E1 -12540.312,E2 -12540.312} C_VEL
LIN {X 0,Y 375.958,Z 348.65,A -85,B 0,C 180,E1 -12544.111,E2 -12544.111} C_VEL
LIN {X 0,Y 375.953,Z 348.654,A -85,B 0,C 180,E1 -12546.74,E2 -12546.74} C_VEL
LIN {X 0,Y 375.993,Z 348.649,A -85,B 0,C 180,E1 -12550.046,E2 -12550.046} C_VEL
LIN {X 0,Y 375.296,Z 348.739,A -85,B 0,C 180,E1 -12550.642,E2 -12550.642} C_VEL
LIN {X 0,Y 372.432,Z 349.095,A -85,B 0,C 180,E1 -12551.574,E2 -12551.574} C_VEL
LIN {X 0,Y 369.585,Z 349.448,A -85,B 0,C 180,E1 -12552.52,E2 -12552.52} C_VEL
LIN {X 0,Y 368.938,Z 349.529,A -85,B 0,C 180,E1 -12553.131,E2 -12553.131} C_VEL
LIN {X 0,Y 369.018,Z 349.75,A -85,B 0,C 180,E1 -12554.02,E2 -12554.02} C_VEL
LIN {X 0,Y 369.339,Z 351.07,A -85,B 0,C 180,E1 -12554.225,E2 -12554.225} C_VEL
LIN {X 0,Y 372.647,Z 362.626,A -85,B 0,C 180,E1 -12555.206,E2 -12555.206} C_VEL
LIN {X 0,Y 373.916,Z 367.573,A -85,B 0,C 180,E1 -12555.685,E2 -12555.685} C_VEL
LIN {X 0,Y 373.174,Z 378.646,A -85,B 0,C 180,E1 -12556.76,E2 -12556.76} C_VEL
LIN {X 0,Y 372.488,Z 388.559,A -85,B 0,C 180,E1 -12557.948,E2 -12557.948} C_VEL
LIN {X 0,Y 371.696,Z 398.272,A -85,B 0,C 180,E1 -12559.376,E2 -12559.376} C_VEL
LIN {X 0,Y 370.919,Z 407.055,A -85,B 0,C 180,E1 -12560.971,E2 -12560.971} C_VEL
LIN {X 0,Y 370.372,Z 414.351,A -85,B 0,C 180,E1 -12562.611,E2 -12562.611} C_VEL
LIN {X 0,Y 369.784,Z 420.738,A -85,B 0,C 180,E1 -12564.428,E2 -12564.428} C_VEL
LIN {X 0,Y 369.396,Z 426.295,A -85,B 0,C 180,E1 -12566.513,E2 -12566.513} C_VEL
LIN {X 0,Y 369.169,Z 428.816,A -85,B 0,C 180,E1 -12567.788,E2 -12567.788} C_VEL
LIN {X 0,Y 369.033,Z 430.784,A -85,B 0,C 180,E1 -12569.056,E2 -12569.056} C_VEL
LIN {X 0,Y 368.946,Z 432.767,A -85,B 0,C 180,E1 -12571.19,E2 -12571.19} C_VEL
LIN {X 0,Y 369.068,Z 433.235,A -85,B 0,C 180,E1 -12573.505,E2 -12573.505} C_VEL
LIN {X 0,Y 369.465,Z 431.8,A -85,B 0,C 180,E1 -12575.929,E2 -12575.929} C_VEL
LIN {X 0,Y 369.897,Z 429.514,A -85,B 0,C 180,E1 -12577.666,E2 -12577.666} C_VEL
LIN {X 0,Y 370.457,Z 425.999,A -85,B 0,C 180,E1 -12579.454,E2 -12579.454} C_VEL
LIN {X 0,Y 371.185,Z 421.241,A -85,B 0,C 180,E1 -12581.223,E2 -12581.223} C_VEL
LIN {X 0,Y 372.029,Z 415.164,A -85,B 0,C 180,E1 -12582.974,E2 -12582.974} C_VEL
LIN {X 0,Y 373.078,Z 407.42,A -85,B 0,C 180,E1 -12584.708,E2 -12584.708} C_VEL
LIN {X 0,Y 374.037,Z 399.49,A -85,B 0,C 180,E1 -12586.139,E2 -12586.139} C_VEL
LIN {X 0,Y 375.154,Z 389.894,A -85,B 0,C 180,E1 -12587.544,E2 -12587.544} C_VEL
LIN {X 0,Y 376.173,Z 378.912,A -85,B 0,C 180,E1 -12588.823,E2 -12588.823} C_VEL
LIN {X 0,Y 376.618,Z 371.627,A -85,B 0,C 180,E1 -12589.54,E2 -12589.54} C_VEL
LIN {X 0,Y 373,Z 360.125,A -85,B 0,C 180,E1 -12590.785,E2 -12590.785} C_VEL
LIN {X 0,Y 369.291,Z 350.178,A -85,B 0,C 180,E1 -12591.773,E2 -12591.773} C_VEL
LIN {X 0,Y 369.178,Z 349.517,A -85,B 0,C 180,E1 -12592.065,E2 -12592.065} C_VEL
LIN {X 0,Y 369.131,Z 349.505,A -85,B 0,C 180,E1 -12594.537,E2 -12594.537} C_VEL
LIN {X 0,Y 369.306,Z 349.485,A -85,B 0,C 180,E1 -12597.819,E2 -12597.819} C_VEL
LIN {X 0,Y 369.448,Z 349.466,A -85,B 0,C 180,E1 -12600,E2 -12600} C_VEL
LIN {X 0,Y 369.307,Z 349.482,A -85,B 0,C 180,E1 -12602.181,E2 -12602.181} C_VEL
LIN {X 0,Y 369.177,Z 349.498,A -85,B 0,C 180,E1 -12606.559,E2 -12606.559} C_VEL
LIN {X 0,Y 369.054,Z 349.512,A -85,B 0,C 180,E1 -12609.869,E2 -12609.869} C_VEL
LIN {X 0,Y 369.029,Z 349.517,A -85,B 0,C 180,E1 -12613.772,E2 -12613.772} C_VEL
LIN {X 0,Y 368.983,Z 349.517,A -85,B 0,C 180,E1 -12617.743,E2 -12617.743} C_VEL
LIN {X 0,Y 368.902,Z 349.53,A -85,B 0,C 180,E1 -12621.221,E2 -12621.221} C_VEL
LIN {X 0,Y 368.947,Z 349.528,A -85,B 0,C 180,E1 -12624.776,E2 -12624.776} C_VEL
LIN {X 0,Y 368.956,Z 349.527,A -85,B 0,C 180,E1 -12627.204,E2 -12627.204} C_VEL
LIN {X 0,Y 368.923,Z 349.529,A -85,B 0,C 180,E1 -12630.954,E2 -12630.954} C_VEL
LIN {X 0,Y 368.923,Z 349.53,A -85,B 0,C 180,E1 -12635.002,E2 -12635.002} C_VEL
LIN {X 0,Y 368.871,Z 349.537,A -85,B 0,C 180,E1 -12638.635,E2 -12638.635} C_VEL
LIN {X 0,Y 368.859,Z 349.54,A -85,B 0,C 180,E1 -12642.007,E2 -12642.007} C_VEL
LIN {X 0,Y 368.922,Z 349.691,A -85,B 0,C 180,E1 -12643.923,E2 -12643.923} C_VEL
LIN {X 0,Y 370.167,Z 355.616,A -85,B 0,C 180,E1 -12646.884,E2 -12646.884} C_VEL
LIN {X 0,Y 371.515,Z 362.532,A -85,B 0,C 180,E1 -12649.972,E2 -12649.972} C_VEL
LIN {X 0,Y 372.542,Z 368.523,A -85,B 0,C 180,E1 -12652.404,E2 -12652.404} C_VEL
LIN {X 0,Y 371.956,Z 373.906,A -85,B 0,C 180,E1 -12654.339,E2 -12654.339} C_VEL
LIN {X 0,Y 370.771,Z 384.485,A -85,B 0,C 180,E1 -12657.945,E2 -12657.945} C_VEL
LIN {X 0,Y 369.826,Z 395.865,A -85,B 0,C 180,E1 -12661.636,E2 -12661.636} C_VEL
LIN {X 0,Y 369.063,Z 407.456,A -85,B 0,C 180,E1 -12665.233,E2 -12665.233} C_VEL
LIN {X 0,Y 368.479,Z 421.033,A -85,B 0,C 180,E1 -12669.322,E2 -12669.322} C_VEL
LIN {X 0,Y 368.541,Z 422.491,A -85,B 0,C 180,E1 -12669.506,E2 -12669.506} C_VEL
LIN {X 0,Y 370.688,Z 435.559,A -85,B 0,C 180,E1 -12670.137,E2 -12670.137} C_VEL
LIN {X 0,Y 371.883,Z 448.494,A -85,B 0,C 180,E1 -12670.896,E2 -12670.896} C_VEL
LIN {X 0,Y 372.163,Z 459.934,A -85,B 0,C 180,E1 -12671.703,E2 -12671.703} C_VEL
LIN {X 0,Y 372.097,Z 471.498,A -85,B 0,C 180,E1 -12672.694,E2 -12672.694} C_VEL
LIN {X 0,Y 371.811,Z 478.443,A -85,B 0,C 180,E1 -12673.388,E2 -12673.388} C_VEL
LIN {X 0,Y 370.429,Z 490.132,A -85,B 0,C 180,E1 -12674.738,E2 -12674.738} C_VEL
LIN {X 0,Y 369.603,Z 499.279,A -85,B 0,C 180,E1 -12676.043,E2 -12676.043} C_VEL
LIN {X 0,Y 368.919,Z 506.931,A -85,B 0,C 180,E1 -12677.345,E2 -12677.345} C_VEL
LIN {X 0,Y 368.331,Z 514.974,A -85,B 0,C 180,E1 -12679,E2 -12679} C_VEL
LIN {X 0,Y 368.031,Z 521.546,A -85,B 0,C 180,E1 -12680.659,E2 -12680.659} C_VEL
LIN {X 0,Y 367.996,Z 526.862,A -85,B 0,C 180,E1 -12682.318,E2 -12682.318} C_VEL
LIN {X 0,Y 368.1,Z 531.025,A -85,B 0,C 180,E1 -12683.972,E2 -12683.972} C_VEL
LIN {X 0,Y 368.296,Z 534.124,A -85,B 0,C 180,E1 -12685.622,E2 -12685.622} C_VEL
LIN {X 0,Y 368.355,Z 535.628,A -85,B 0,C 180,E1 -12686.719,E2 -12686.719} C_VEL
LIN {X 0,Y 368.406,Z 536.703,A -85,B 0,C 180,E1 -12687.813,E2 -12687.813} C_VEL
LIN {X 0,Y 368.715,Z 537.346,A -85,B 0,C 180,E1 -12688.908,E2 -12688.908} C_VEL
LIN {X 0,Y 368.787,Z 537.539,A -85,B 0,C 180,E1 -12690,E2 -12690} C_VEL
LIN {X 0,Y 368.712,Z 537.301,A -85,B 0,C 180,E1 -12691.092,E2 -12691.092} C_VEL
LIN {X 0,Y 368.427,Z 536.599,A -85,B 0,C 180,E1 -12692.186,E2 -12692.186} C_VEL
LIN {X 0,Y 368.387,Z 535.463,A -85,B 0,C 180,E1 -12693.281,E2 -12693.281} C_VEL
LIN {X 0,Y 368.276,Z 532.934,A -85,B 0,C 180,E1 -12694.926,E2 -12694.926} C_VEL
LIN {X 0,Y 368.109,Z 528.527,A -85,B 0,C 180,E1 -12696.881,E2 -12696.881} C_VEL
LIN {X 0,Y 368.066,Z 522.673,A -85,B 0,C 180,E1 -12698.786,E2 -12698.786} C_VEL
LIN {X 0,Y 368.223,Z 516.1,A -85,B 0,C 180,E1 -12700.446,E2 -12700.446} C_VEL
LIN {X 0,Y 368.727,Z 507.959,A -85,B 0,C 180,E1 -12702.102,E2 -12702.102} C_VEL
LIN {X 0,Y 369.308,Z 500.015,A -85,B 0,C 180,E1 -12703.424,E2 -12703.424} C_VEL
LIN {X 0,Y 370.151,Z 489.5,A -85,B 0,C 180,E1 -12704.852,E2 -12704.852} C_VEL
LIN {X 0,Y 371.173,Z 478.197,A -85,B 0,C 180,E1 -12706.076,E2 -12706.076} C_VEL
LIN {X 0,Y 371.453,Z 472.193,A -85,B 0,C 180,E1 -12706.628,E2 -12706.628} C_VEL
LIN {X 0,Y 370.976,Z 460.065,A -85,B 0,C 180,E1 -12707.573,E2 -12707.573} C_VEL
LIN {X 0,Y 370.063,Z 446.933,A -85,B 0,C 180,E1 -12708.372,E2 -12708.372} C_VEL
LIN {X 0,Y 368.836,Z 433.32,A -85,B 0,C 180,E1 -12708.972,E2 -12708.972} C_VEL
LIN {X 0,Y 368.374,Z 428.559,A -85,B 0,C 180,E1 -12709.178,E2 -12709.178} C_VEL
LIN {X 0,Y 368.47,Z 425.302,A -85,B 0,C 180,E1 -12710.079,E2 -12710.079} C_VEL
LIN {X 0,Y 369.13,Z 412.625,A -85,B 0,C 180,E1 -12713.951,E2 -12713.951} C_VEL
LIN {X 0,Y 369.959,Z 400.468,A -85,B 0,C 180,E1 -12717.737,E2 -12717.737} C_VEL
LIN {X 0,Y 371.174,Z 386.93,A -85,B 0,C 180,E1 -12722.016,E2 -12722.016} C_VEL
LIN {X 0,Y 372.692,Z 373.302,A -85,B 0,C 180,E1 -12726.441,E2 -12726.441} C_VEL
LIN {X 0,Y 372.831,Z 369.682,A -85,B 0,C 180,E1 -12727.654,E2 -12727.654} C_VEL
LIN {X 0,Y 370.913,Z 359.829,A -85,B 0,C 180,E1 -12731.233,E2 -12731.233} C_VEL
LIN {X 0,Y 368.978,Z 349.653,A -85,B 0,C 180,E1 -12735.155,E2 -12735.155} C_VEL
LIN {X 0,Y 368.864,Z 349.535,A -85,B 0,C 180,E1 -12738.175,E2 -12738.175} C_VEL
LIN {X 0,Y 368.871,Z 349.54,A -85,B 0,C 180,E1 -12741.365,E2 -12741.365} C_VEL
LIN {X 0,Y 368.93,Z 349.531,A -85,B 0,C 180,E1 -12745.146,E2 -12745.146} C_VEL
LIN {X 0,Y 368.923,Z 349.531,A -85,B 0,C 180,E1 -12749.046,E2 -12749.046} C_VEL
LIN {X 0,Y 368.969,Z 349.524,A -85,B 0,C 180,E1 -12751.563,E2 -12751.563} C_VEL
LIN {X 0,Y 368.992,Z 349.518,A -85,B 0,C 180,E1 -12754.019,E2 -12754.019} C_VEL
LIN {X 0,Y 368.914,Z 349.53,A -85,B 0,C 180,E1 -12757.604,E2 -12757.604} C_VEL
LIN {X 0,Y 368.946,Z 349.53,A -85,B 0,C 180,E1 -12761.105,E2 -12761.105} C_VEL
LIN {X 0,Y 368.988,Z 349.52,A -85,B 0,C 180,E1 -12764.535,E2 -12764.535} C_VEL
LIN {X 0,Y 368.995,Z 349.518,A -85,B 0,C 180,E1 -12767.906,E2 -12767.906} C_VEL
LIN {X 0,Y 369.137,Z 349.5,A -85,B 0,C 180,E1 -12771.891,E2 -12771.891} C_VEL
LIN {X 0,Y 369.128,Z 349.504,A -85,B 0,C 180,E1 -12774.537,E2 -12774.537} C_VEL
LIN {X 0,Y 369.306,Z 349.479,A -85,B 0,C 180,E1 -12777.819,E2 -12777.819} C_VEL
LIN {X 0,Y 369.448,Z 349.461,A -85,B 0,C 180,E1 -12780,E2 -12780} C_VEL
LIN {X 0,Y 369.306,Z 349.48,A -85,B 0,C 180,E1 -12782.181,E2 -12782.181} C_VEL
LIN {X 0,Y 369.181,Z 349.498,A -85,B 0,C 180,E1 -12786.674,E2 -12786.674} C_VEL
LIN {X 0,Y 369.058,Z 349.51,A -85,B 0,C 180,E1 -12789.868,E2 -12789.868} C_VEL
LIN {X 0,Y 369.029,Z 349.514,A -85,B 0,C 180,E1 -12793.772,E2 -12793.772} C_VEL
LIN {X 0,Y 368.993,Z 349.518,A -85,B 0,C 180,E1 -12797.769,E2 -12797.769} C_VEL
LIN {X 0,Y 368.922,Z 349.527,A -85,B 0,C 180,E1 -12801.22,E2 -12801.22} C_VEL
LIN {X 0,Y 368.95,Z 349.526,A -85,B 0,C 180,E1 -12804.776,E2 -12804.776} C_VEL
LIN {X 0,Y 368.98,Z 349.526,A -85,B 0,C 180,E1 -12808.436,E2 -12808.436} C_VEL
LIN {X 0,Y 368.893,Z 349.536,A -85,B 0,C 180,E1 -12812.239,E2 -12812.239} C_VEL
LIN {X 0,Y 368.923,Z 349.527,A -85,B 0,C 180,E1 -12815.002,E2 -12815.002} C_VEL
LIN {X 0,Y 368.907,Z 349.531,A -85,B 0,C 180,E1 -12818.642,E2 -12818.642} C_VEL
LIN {X 0,Y 368.905,Z 349.531,A -85,B 0,C 180,E1 -12821.819,E2 -12821.819} C_VEL
LIN {X 0,Y 368.877,Z 349.532,A -85,B 0,C 180,E1 -12825.177,E2 -12825.177} C_VEL
LIN {X 0,Y 368.885,Z 349.538,A -85,B 0,C 180,E1 -12828.179,E2 -12828.179} C_VEL
LIN {X 0,Y 368.907,Z 349.529,A -85,B 0,C 180,E1 -12831.36,E2 -12831.36} C_VEL
LIN {X 0,Y 368.935,Z 349.525,A -85,B 0,C 180,E1 -12835.147,E2 -12835.147} C_VEL
LIN {X 0,Y 368.928,Z 349.526,A -85,B 0,C 180,E1 -12839.047,E2 -12839.047} C_VEL
LIN {X 0,Y 368.986,Z 349.521,A -85,B 0,C 180,E1 -12841.565,E2 -12841.565} C_VEL
LIN {X 0,Y 368.958,Z 349.523,A -85,B 0,C 180,E1 -12845.225,E2 -12845.225} C_VEL
LIN {X 0,Y 368.938,Z 349.525,A -85,B 0,C 180,E1 -12848.974,E2 -12848.974} C_VEL
LIN {X 0,Y 368.992,Z 349.52,A -85,B 0,C 180,E1 -12852.258,E2 -12852.258} C_VEL
LIN {X 0,Y 369.018,Z 349.521,A -85,B 0,C 180,E1 -12855.666,E2 -12855.666} C_VEL
LIN {X 0,Y 369.024,Z 349.515,A -85,B 0,C 180,E1 -12859.021,E2 -12859.021} C_VEL
LIN {X 0,Y 369.191,Z 349.494,A -85,B 0,C 180,E1 -12862.343,E2 -12862.343} C_VEL
LIN {X 0,Y 369.148,Z 349.499,A -85,B 0,C 180,E1 -12864.538,E2 -12864.538} C_VEL
LIN {X 0,Y 369.321,Z 349.481,A -85,B 0,C 180,E1 -12867.819,E2 -12867.819} C_VEL
LIN {X 0,Y 369.461,Z 349.462,A -85,B 0,C 180,E1 -12870,E2 -12870} C_VEL
LIN {X 0,Y 369.322,Z 349.478,A -85,B 0,C 180,E1 -12872.181,E2 -12872.181} C_VEL
LIN {X 0,Y 369.201,Z 349.492,A -85,B 0,C 180,E1 -12876.558,E2 -12876.558} C_VEL
LIN {X 0,Y 369.07,Z 349.51,A -85,B 0,C 180,E1 -12879.868,E2 -12879.868} C_VEL
LIN {X 0,Y 369.038,Z 349.515,A -85,B 0,C 180,E1 -12883.772,E2 -12883.772} C_VEL
LIN {X 0,Y 369.002,Z 349.519,A -85,B 0,C 180,E1 -12887.768,E2 -12887.768} C_VEL
LIN {X 0,Y 368.929,Z 349.532,A -85,B 0,C 180,E1 -12891.219,E2 -12891.219} C_VEL
LIN {X 0,Y 368.958,Z 349.525,A -85,B 0,C 180,E1 -12894.775,E2 -12894.775} C_VEL
LIN {X 0,Y 368.962,Z 349.528,A -85,B 0,C 180,E1 -12897.203,E2 -12897.203} C_VEL
LIN {X 0,Y 368.928,Z 349.531,A -85,B 0,C 180,E1 -12900.953,E2 -12900.953} C_VEL
LIN {X 0,Y 368.927,Z 349.532,A -85,B 0,C 180,E1 -12905.001,E2 -12905.001} C_VEL
LIN {X 0,Y 368.911,Z 349.531,A -85,B 0,C 180,E1 -12908.641,E2 -12908.641} C_VEL
LIN {X 0,Y 368.939,Z 349.529,A -85,B 0,C 180,E1 -12912.019,E2 -12912.019} C_VEL
LIN {X 0,Y 368.938,Z 349.529,A -85,B 0,C 180,E1 -12913.131,E2 -12913.131} C_VEL
LIN {X 0,Y 368.916,Z 350.274,A -85,B 0,C 180,E1 -12913.577,E2 -12913.577} C_VEL
LIN {X 0,Y 368.774,Z 352.773,A -85,B 0,C 180,E1 -12914.074,E2 -12914.074} C_VEL
LIN {X 0,Y 368.457,Z 357.25,A -85,B 0,C 180,E1 -12914.557,E2 -12914.557} C_VEL
LIN {X 0,Y 367.333,Z 368.316,A -85,B 0,C 180,E1 -12915.444,E2 -12915.444} C_VEL
LIN {X 0,Y 366.643,Z 374.992,A -85,B 0,C 180,E1 -12916.062,E2 -12916.062} C_VEL
LIN {X 0,Y 365.897,Z 385.69,A -85,B 0,C 180,E1 -12917.259,E2 -12917.259} C_VEL
LIN {X 0,Y 365.062,Z 395.776,A -85,B 0,C 180,E1 -12918.659,E2 -12918.659} C_VEL
LIN {X 0,Y 364.319,Z 404.284,A -85,B 0,C 180,E1 -12920.102,E2 -12920.102} C_VEL
LIN {X 0,Y 363.563,Z 412.407,A -85,B 0,C 180,E1 -12921.787,E2 -12921.787} C_VEL
LIN {X 0,Y 363.054,Z 418.858,A -85,B 0,C 180,E1 -12923.469,E2 -12923.469} C_VEL
LIN {X 0,Y 362.567,Z 423.947,A -85,B 0,C 180,E1 -12925.122,E2 -12925.122} C_VEL
LIN {X 0,Y 362.243,Z 428.567,A -85,B 0,C 180,E1 -12927.096,E2 -12927.096} C_VEL
LIN {X 0,Y 362.021,Z 431.231,A -85,B 0,C 180,E1 -12928.667,E2 -12928.667} C_VEL
LIN {X 0,Y 361.949,Z 432.508,A -85,B 0,C 180,E1 -12929.679,E2 -12929.679} C_VEL
LIN {X 0,Y 361.937,Z 433.632,A -85,B 0,C 180,E1 -12930.958,E2 -12930.958} C_VEL
LIN {X 0,Y 361.961,Z 434.214,A -85,B 0,C 180,E1 -12932.225,E2 -12932.225} C_VEL
LIN {X 0,Y 362.073,Z 434.306,A -85,B 0,C 180,E1 -12933.484,E2 -12933.484} C_VEL
LIN {X 0,Y 362.404,Z 433.172,A -85,B 0,C 180,E1 -12935.704,E2 -12935.704} C_VEL
LIN {X 0,Y 362.773,Z 431.503,A -85,B 0,C 180,E1 -12937.203,E2 -12937.203} C_VEL
LIN {X 0,Y 363.342,Z 428.422,A -85,B 0,C 180,E1 -12939.032,E2 -12939.032} C_VEL
LIN {X 0,Y 364.119,Z 423.628,A -85,B 0,C 180,E1 -12941.04,E2 -12941.04} C_VEL
LIN {X 0,Y 365.063,Z 417.483,A -85,B 0,C 180,E1 -12942.927,E2 -12942.927} C_VEL
LIN {X 0,Y 366.147,Z 410.106,A -85,B 0,C 180,E1 -12944.697,E2 -12944.697} C_VEL
LIN {X 0,Y 367.182,Z 402.491,A -85,B 0,C 180,E1 -12946.157,E2 -12946.157} C_VEL
LIN {X 0,Y 368.244,Z 393.801,A -85,B 0,C 180,E1 -12947.516,E2 -12947.516} C_VEL
LIN {X 0,Y 369.391,Z 382.938,A -85,B 0,C 180,E1 -12948.893,E2 -12948.893} C_VEL
LIN {X 0,Y 370.055,Z 373.438,A -85,B 0,C 180,E1 -12949.882,E2 -12949.882} C_VEL
LIN {X 0,Y 366.465,Z 362.021,A -85,B 0,C 180,E1 -12951.175,E2 -12951.175} C_VEL
LIN {X 0,Y 362.233,Z 350.987,A -85,B 0,C 180,E1 -12952.335,E2 -12952.335} C_VEL
LIN {X 0,Y 362.123,Z 350.397,A -85,B 0,C 180,E1 -12952.613,E2 -12952.613} C_VEL
LIN {X 0,Y 362.105,Z 350.381,A -85,B 0,C 180,E1 -12954.431,E2 -12954.431} C_VEL
LIN {X 0,Y 362.27,Z 350.362,A -85,B 0,C 180,E1 -12957.776,E2 -12957.776} C_VEL
LIN {X 0,Y 362.418,Z 350.342,A -85,B 0,C 180,E1 -12960,E2 -12960} C_VEL
LIN {X 0,Y 362.271,Z 350.358,A -85,B 0,C 180,E1 -12962.224,E2 -12962.224} C_VEL
LIN {X 0,Y 362.138,Z 350.375,A -85,B 0,C 180,E1 -12966.687,E2 -12966.687} C_VEL
LIN {X 0,Y 361.991,Z 350.391,A -85,B 0,C 180,E1 -12970.063,E2 -12970.063} C_VEL
LIN {X 0,Y 361.99,Z 350.393,A -85,B 0,C 180,E1 -12973.899,E2 -12973.899} C_VEL
LIN {X 0,Y 361.92,Z 350.4,A -85,B 0,C 180,E1 -12976.935,E2 -12976.935} C_VEL
LIN {X 0,Y 361.875,Z 350.404,A -85,B 0,C 180,E1 -12980.462,E2 -12980.462} C_VEL
LIN {X 0,Y 361.886,Z 350.403,A -85,B 0,C 180,E1 -12984.113,E2 -12984.113} C_VEL
LIN {X 0,Y 361.934,Z 350.398,A -85,B 0,C 180,E1 -12986.722,E2 -12986.722} C_VEL
LIN {X 0,Y 361.866,Z 350.411,A -85,B 0,C 180,E1 -12990.329,E2 -12990.329} C_VEL
LIN {X 0,Y 361.848,Z 350.413,A -85,B 0,C 180,E1 -12994.281,E2 -12994.281} C_VEL
LIN {X 0,Y 361.854,Z 350.411,A -85,B 0,C 180,E1 -12997.223,E2 -12997.223} C_VEL
LIN {X 0,Y 361.806,Z 350.419,A -85,B 0,C 180,E1 -13000.752,E2 -13000.752} C_VEL
LIN {X 0,Y 361.876,Z 350.652,A -85,B 0,C 180,E1 -13003.321,E2 -13003.321} C_VEL
LIN {X 0,Y 363.201,Z 356.796,A -85,B 0,C 180,E1 -13006.521,E2 -13006.521} C_VEL
LIN {X 0,Y 364.588,Z 363.899,A -85,B 0,C 180,E1 -13009.779,E2 -13009.779} C_VEL
LIN {X 0,Y 365.552,Z 369.267,A -85,B 0,C 180,E1 -13012.033,E2 -13012.033} C_VEL
LIN {X 0,Y 365.624,Z 371.061,A -85,B 0,C 180,E1 -13012.737,E2 -13012.737} C_VEL
LIN {X 0,Y 364.173,Z 382.075,A -85,B 0,C 180,E1 -13016.654,E2 -13016.654} C_VEL
LIN {X 0,Y 363.119,Z 392.713,A -85,B 0,C 180,E1 -13020.252,E2 -13020.252} C_VEL
LIN {X 0,Y 362.236,Z 404.701,A -85,B 0,C 180,E1 -13024.118,E2 -13024.118} C_VEL
LIN {X 0,Y 361.572,Z 416.303,A -85,B 0,C 180,E1 -13027.727,E2 -13027.727} C_VEL
LIN {X 0,Y 361.464,Z 420.259,A -85,B 0,C 180,E1 -13028.876,E2 -13028.876} C_VEL
LIN {X 0,Y 362.02,Z 423.569,A -85,B 0,C 180,E1 -13029.088,E2 -13029.088} C_VEL
LIN {X 0,Y 364.114,Z 437.015,A -85,B 0,C 180,E1 -13029.792,E2 -13029.792} C_VEL
LIN {X 0,Y 365.165,Z 449.5,A -85,B 0,C 180,E1 -13030.572,E2 -13030.572} C_VEL
LIN {X 0,Y 365.354,Z 461.727,A -85,B 0,C 180,E1 -13031.499,E2 -13031.499} C_VEL
LIN {X 0,Y 365.212,Z 474.028,A -85,B 0,C 180,E1 -13032.646,E2 -13032.646} C_VEL
LIN {X 0,Y 364.355,Z 482.903,A -85,B 0,C 180,E1 -13033.615,E2 -13033.615} C_VEL
LIN {X 0,Y 363.282,Z 492.517,A -85,B 0,C 180,E1 -13034.861,E2 -13034.861} C_VEL
LIN {X 0,Y 362.52,Z 500.879,A -85,B 0,C 180,E1 -13036.157,E2 -13036.157} C_VEL
LIN {X 0,Y 361.692,Z 509.012,A -85,B 0,C 180,E1 -13037.659,E2 -13037.659} C_VEL
LIN {X 0,Y 361.128,Z 516.496,A -85,B 0,C 180,E1 -13039.346,E2 -13039.346} C_VEL
LIN {X 0,Y 360.913,Z 522.58,A -85,B 0,C 180,E1 -13041.038,E2 -13041.038} C_VEL
LIN {X 0,Y 360.942,Z 527.596,A -85,B 0,C 180,E1 -13042.785,E2 -13042.785} C_VEL
LIN {X 0,Y 361.041,Z 531.221,A -85,B 0,C 180,E1 -13044.415,E2 -13044.415} C_VEL
LIN {X 0,Y 361.225,Z 533.155,A -85,B 0,C 180,E1 -13045.537,E2 -13045.537} C_VEL
LIN {X 0,Y 361.304,Z 534.652,A -85,B 0,C 180,E1 -13046.655,E2 -13046.655} C_VEL
LIN {X 0,Y 361.363,Z 535.703,A -85,B 0,C 180,E1 -13047.771,E2 -13047.771} C_VEL
LIN {X 0,Y 361.683,Z 536.331,A -85,B 0,C 180,E1 -13048.887,E2 -13048.887} C_VEL
LIN {X 0,Y 361.785,Z 536.519,A -85,B 0,C 180,E1 -13050,E2 -13050} C_VEL
LIN {X 0,Y 361.682,Z 536.265,A -85,B 0,C 180,E1 -13051.113,E2 -13051.113} C_VEL
LIN {X 0,Y 361.393,Z 535.528,A -85,B 0,C 180,E1 -13052.229,E2 -13052.229} C_VEL
LIN {X 0,Y 361.35,Z 534.375,A -85,B 0,C 180,E1 -13053.345,E2 -13053.345} C_VEL
LIN {X 0,Y 361.221,Z 531.807,A -85,B 0,C 180,E1 -13055.023,E2 -13055.023} C_VEL
LIN {X 0,Y 361.043,Z 527.658,A -85,B 0,C 180,E1 -13056.899,E2 -13056.899} C_VEL
LIN {X 0,Y 360.999,Z 523.314,A -85,B 0,C 180,E1 -13058.396,E2 -13058.396} C_VEL
LIN {X 0,Y 361.09,Z 517.182,A -85,B 0,C 180,E1 -13060.088,E2 -13060.088} C_VEL
LIN {X 0,Y 361.542,Z 509.57,A -85,B 0,C 180,E1 -13061.777,E2 -13061.777} C_VEL
LIN {X 0,Y 362.22,Z 500.009,A -85,B 0,C 180,E1 -13063.463,E2 -13063.463} C_VEL
LIN {X 0,Y 363.023,Z 490.212,A -85,B 0,C 180,E1 -13064.863,E2 -13064.863} C_VEL
LIN {X 0,Y 363.993,Z 479.286,A -85,B 0,C 180,E1 -13066.114,E2 -13066.114} C_VEL
LIN {X 0,Y 364.449,Z 473.546,A -85,B 0,C 180,E1 -13066.669,E2 -13066.669} C_VEL
LIN {X 0,Y 364.036,Z 461.217,A -85,B 0,C 180,E1 -13067.702,E2 -13067.702} C_VEL
LIN {X 0,Y 363.195,Z 448.54,A -85,B 0,C 180,E1 -13068.526,E2 -13068.526} C_VEL
LIN {X 0,Y 361.98,Z 434.309,A -85,B 0,C 180,E1 -13069.211,E2 -13069.211} C_VEL
LIN {X 0,Y 361.322,Z 427.543,A -85,B 0,C 180,E1 -13069.493,E2 -13069.493} C_VEL
LIN {X 0,Y 361.968,Z 414.687,A -85,B 0,C 180,E1 -13073.454,E2 -13073.454} C_VEL
LIN {X 0,Y 362.774,Z 402.613,A -85,B 0,C 180,E1 -13077.275,E2 -13077.275} C_VEL
LIN {X 0,Y 363.719,Z 391.679,A -85,B 0,C 180,E1 -13080.8,E2 -13080.8} C_VEL
LIN {X 0,Y 364.899,Z 380.038,A -85,B 0,C 180,E1 -13084.621,E2 -13084.621} C_VEL
LIN {X 0,Y 365.878,Z 372.245,A -85,B 0,C 180,E1 -13087.233,E2 -13087.233} C_VEL
LIN {X 0,Y 365.109,Z 367.128,A -85,B 0,C 180,E1 -13089.079,E2 -13089.079} C_VEL
LIN {X 0,Y 363.256,Z 357.618,A -85,B 0,C 180,E1 -13092.676,E2 -13092.676} C_VEL
LIN {X 0,Y 361.884,Z 350.484,A -85,B 0,C 180,E1 -13095.544,E2 -13095.544} C_VEL
LIN {X 0,Y 361.807,Z 350.418,A -85,B 0,C 180,E1 -13099.248,E2 -13099.248} C_VEL
LIN {X 0,Y 361.858,Z 350.41,A -85,B 0,C 180,E1 -13102.981,E2 -13102.981} C_VEL
LIN {X 0,Y 361.852,Z 350.408,A -85,B 0,C 180,E1 -13106.63,E2 -13106.63} C_VEL
LIN {X 0,Y 361.868,Z 350.408,A -85,B 0,C 180,E1 -13109.671,E2 -13109.671} C_VEL
LIN {X 0,Y 361.947,Z 350.399,A -85,B 0,C 180,E1 -13113.474,E2 -13113.474} C_VEL
LIN {X 0,Y 361.871,Z 350.412,A -85,B 0,C 180,E1 -13117.143,E2 -13117.143} C_VEL
LIN {X 0,Y 361.877,Z 350.407,A -85,B 0,C 180,E1 -13120.722,E2 -13120.722} C_VEL
LIN {X 0,Y 361.934,Z 350.398,A -85,B 0,C 180,E1 -13124.226,E2 -13124.226} C_VEL
LIN {X 0,Y 361.99,Z 350.392,A -85,B 0,C 180,E1 -13126.527,E2 -13126.527} C_VEL
LIN {X 0,Y 361.991,Z 350.39,A -85,B 0,C 180,E1 -13129.937,E2 -13129.937} C_VEL
LIN {X 0,Y 362.138,Z 350.374,A -85,B 0,C 180,E1 -13133.313,E2 -13133.313} C_VEL
LIN {X 0,Y 362.27,Z 350.355,A -85,B 0,C 180,E1 -13137.776,E2 -13137.776} C_VEL
LIN {X 0,Y 362.418,Z 350.337,A -85,B 0,C 180,E1 -13140,E2 -13140} C_VEL
LIN {X 0,Y 362.27,Z 350.357,A -85,B 0,C 180,E1 -13142.224,E2 -13142.224} C_VEL
LIN {X 0,Y 362.153,Z 350.376,A -85,B 0,C 180,E1 -13146.686,E2 -13146.686} C_VEL
LIN {X 0,Y 362.056,Z 350.386,A -85,B 0,C 180,E1 -13148.934,E2 -13148.934} C_VEL
LIN {X 0,Y 361.951,Z 350.398,A -85,B 0,C 180,E1 -13152.333,E2 -13152.333} C_VEL
LIN {X 0,Y 361.954,Z 350.401,A -85,B 0,C 180,E1 -13154.621,E2 -13154.621} C_VEL
LIN {X 0,Y 361.952,Z 350.397,A -85,B 0,C 180,E1 -13158.1,E2 -13158.1} C_VEL
LIN {X 0,Y 361.885,Z 350.404,A -85,B 0,C 180,E1 -13161.653,E2 -13161.653} C_VEL
LIN {X 0,Y 361.921,Z 350.399,A -85,B 0,C 180,E1 -13165.291,E2 -13165.291} C_VEL
LIN {X 0,Y 361.916,Z 350.4,A -85,B 0,C 180,E1 -13167.778,E2 -13167.778} C_VEL
LIN {X 0,Y 361.84,Z 350.409,A -85,B 0,C 180,E1 -13171.286,E2 -13171.286} C_VEL
LIN {X 0,Y 361.848,Z 350.414,A -85,B 0,C 180,E1 -13174.281,E2 -13174.281} C_VEL
LIN {X 0,Y 361.86,Z 350.407,A -85,B 0,C 180,E1 -13177.224,E2 -13177.224} C_VEL
LIN {X 0,Y 361.868,Z 350.407,A -85,B 0,C 180,E1 -13180.763,E2 -13180.763} C_VEL
LIN {X 0,Y 361.819,Z 350.416,A -85,B 0,C 180,E1 -13184.368,E2 -13184.368} C_VEL
LIN {X 0,Y 361.84,Z 350.41,A -85,B 0,C 180,E1 -13187.568,E2 -13187.568} C_VEL
LIN {X 0,Y 361.868,Z 350.406,A -85,B 0,C 180,E1 -13190.974,E2 -13190.974} C_VEL
LIN {X 0,Y 361.873,Z 350.406,A -85,B 0,C 180,E1 -13194.656,E2 -13194.656} C_VEL
LIN {X 0,Y 361.858,Z 350.409,A -85,B 0,C 180,E1 -13198.374,E2 -13198.374} C_VEL
LIN {X 0,Y 361.922,Z 350.402,A -85,B 0,C 180,E1 -13202.223,E2 -13202.223} C_VEL
LIN {X 0,Y 361.928,Z 350.398,A -85,B 0,C 180,E1 -13204.711,E2 -13204.711} C_VEL
LIN {X 0,Y 361.892,Z 350.404,A -85,B 0,C 180,E1 -13208.348,E2 -13208.348} C_VEL
LIN {X 0,Y 361.969,Z 350.397,A -85,B 0,C 180,E1 -13212.062,E2 -13212.062} C_VEL
LIN {X 0,Y 361.999,Z 350.392,A -85,B 0,C 180,E1 -13216.102,E2 -13216.102} C_VEL
LIN {X 0,Y 362.033,Z 350.389,A -85,B 0,C 180,E1 -13219.938,E2 -13219.938} C_VEL
LIN {X 0,Y 362.154,Z 350.371,A -85,B 0,C 180,E1 -13222.193,E2 -13222.193} C_VEL
LIN {X 0,Y 362.121,Z 350.374,A -85,B 0,C 180,E1 -13224.431,E2 -13224.431} C_VEL
LIN {X 0,Y 362.285,Z 350.358,A -85,B 0,C 180,E1 -13227.777,E2 -13227.777} C_VEL
LIN {X 0,Y 362.431,Z 350.337,A -85,B 0,C 180,E1 -13230,E2 -13230} C_VEL
LIN {X 0,Y 362.286,Z 350.354,A -85,B 0,C 180,E1 -13232.223,E2 -13232.223} C_VEL
LIN {X 0,Y 362.163,Z 350.369,A -85,B 0,C 180,E1 -13236.686,E2 -13236.686} C_VEL
LIN {X 0,Y 362.033,Z 350.386,A -85,B 0,C 180,E1 -13240.062,E2 -13240.062} C_VEL
LIN {X 0,Y 361.999,Z 350.391,A -85,B 0,C 180,E1 -13243.898,E2 -13243.898} C_VEL
LIN {X 0,Y 361.968,Z 350.394,A -85,B 0,C 180,E1 -13247.938,E2 -13247.938} C_VEL
LIN {X 0,Y 361.892,Z 350.405,A -85,B 0,C 180,E1 -13251.652,E2 -13251.652} C_VEL
LIN {X 0,Y 361.928,Z 350.403,A -85,B 0,C 180,E1 -13255.289,E2 -13255.289} C_VEL
LIN {X 0,Y 361.908,Z 350.402,A -85,B 0,C 180,E1 -13257.778,E2 -13257.778} C_VEL
LIN {X 0,Y 361.836,Z 350.411,A -85,B 0,C 180,E1 -13261.629,E2 -13261.629} C_VEL
LIN {X 0,Y 361.873,Z 350.408,A -85,B 0,C 180,E1 -13265.344,E2 -13265.344} C_VEL
LIN {X 0,Y 361.873,Z 350.411,A -85,B 0,C 180,E1 -13269.027,E2 -13269.027} C_VEL
LIN {X 0,Y 361.884,Z 350.407,A -85,B 0,C 180,E1 -13272.44,E2 -13272.44} C_VEL
LIN {X 0,Y 361.966,Z 350.596,A -85,B 0,C 180,E1 -13273.725,E2 -13273.725} C_VEL
LIN {X 0,Y 362.265,Z 351.885,A -85,B 0,C 180,E1 -13273.937,E2 -13273.937} C_VEL
LIN {X 0,Y 365.597,Z 363.505,A -85,B 0,C 180,E1 -13274.946,E2 -13274.946} C_VEL
LIN {X 0,Y 367.027,Z 369.361,A -85,B 0,C 180,E1 -13275.527,E2 -13275.527} C_VEL
LIN {X 0,Y 366.643,Z 374.992,A -85,B 0,C 180,E1 -13276.062,E2 -13276.062} C_VEL
LIN {X 0,Y 365.632,Z 379.943,A -85,B 0,C 180,E1 -13276.546,E2 -13276.546} C_VEL
LIN {X 0,Y 362.243,Z 387.807,A -85,B 0,C 180,E1 -13277.342,E2 -13277.342} C_VEL
LIN {X 0,Y 358.858,Z 395.182,A -85,B 0,C 180,E1 -13278.246,E2 -13278.246} C_VEL
LIN {X 0,Y 357.866,Z 399.364,A -85,B 0,C 180,E1 -13278.893,E2 -13278.893} C_VEL
LIN {X 0,Y 357.064,Z 408.147,A -85,B 0,C 180,E1 -13280.516,E2 -13280.516} C_VEL
LIN {X 0,Y 356.408,Z 416.008,A -85,B 0,C 180,E1 -13282.317,E2 -13282.317} C_VEL
LIN {X 0,Y 355.843,Z 422.103,A -85,B 0,C 180,E1 -13284.071,E2 -13284.071} C_VEL
LIN {X 0,Y 355.385,Z 427.642,A -85,B 0,C 180,E1 -13286.156,E2 -13286.156} C_VEL
LIN {X 0,Y 355.054,Z 431.765,A -85,B 0,C 180,E1 -13288.335,E2 -13288.335} C_VEL
LIN {X 0,Y 354.922,Z 434.364,A -85,B 0,C 180,E1 -13290.604,E2 -13290.604} C_VEL
LIN {X 0,Y 354.911,Z 435.021,A -85,B 0,C 180,E1 -13291.624,E2 -13291.624} C_VEL
LIN {X 0,Y 355.01,Z 435.356,A -85,B 0,C 180,E1 -13292.977,E2 -13292.977} C_VEL
LIN {X 0,Y 355.155,Z 435.2,A -85,B 0,C 180,E1 -13294.192,E2 -13294.192} C_VEL
LIN {X 0,Y 355.356,Z 434.545,A -85,B 0,C 180,E1 -13295.469,E2 -13295.469} C_VEL
LIN {X 0,Y 355.655,Z 433.385,A -85,B 0,C 180,E1 -13296.721,E2 -13296.721} C_VEL
LIN {X 0,Y 356.256,Z 430.63,A -85,B 0,C 180,E1 -13298.651,E2 -13298.651} C_VEL
LIN {X 0,Y 356.882,Z 426.925,A -85,B 0,C 180,E1 -13300.441,E2 -13300.441} C_VEL
LIN {X 0,Y 357.779,Z 421.785,A -85,B 0,C 180,E1 -13302.274,E2 -13302.274} C_VEL
LIN {X 0,Y 358.807,Z 415.237,A -85,B 0,C 180,E1 -13304.084,E2 -13304.084} C_VEL
LIN {X 0,Y 360.058,Z 406.993,A -85,B 0,C 180,E1 -13305.878,E2 -13305.878} C_VEL
LIN {X 0,Y 361.252,Z 398.366,A -85,B 0,C 180,E1 -13307.374,E2 -13307.374} C_VEL
LIN {X 0,Y 362.348,Z 389.2,A -85,B 0,C 180,E1 -13308.675,E2 -13308.675} C_VEL
LIN {X 0,Y 363.385,Z 379.174,A -85,B 0,C 180,E1 -13309.835,E2 -13309.835} C_VEL
LIN {X 0,Y 363.644,Z 376.261,A -85,B 0,C 180,E1 -13310.124,E2 -13310.124} C_VEL
LIN {X 0,Y 360.831,Z 366.656,A -85,B 0,C 180,E1 -13311.277,E2 -13311.277} C_VEL
LIN {X 0,Y 357.174,Z 356.723,A -85,B 0,C 180,E1 -13312.368,E2 -13312.368} C_VEL
LIN {X 0,Y 355.195,Z 351.91,A -85,B 0,C 180,E1 -13312.896,E2 -13312.896} C_VEL
LIN {X 0,Y 355.118,Z 351.275,A -85,B 0,C 180,E1 -13313.18,E2 -13313.18} C_VEL
LIN {X 0,Y 355.233,Z 351.238,A -85,B 0,C 180,E1 -13317.732,E2 -13317.732} C_VEL
LIN {X 0,Y 355.388,Z 351.218,A -85,B 0,C 180,E1 -13320,E2 -13320} C_VEL
LIN {X 0,Y 355.234,Z 351.235,A -85,B 0,C 180,E1 -13322.268,E2 -13322.268} C_VEL
LIN {X 0,Y 355.102,Z 351.252,A -85,B 0,C 180,E1 -13326.82,E2 -13326.82} C_VEL
LIN {X 0,Y 354.947,Z 351.269,A -85,B 0,C 180,E1 -13330.265,E2 -13330.265} C_VEL
LIN {X 0,Y 354.934,Z 351.272,A -85,B 0,C 180,E1 -13334.019,E2 -13334.019} C_VEL
LIN {X 0,Y 354.882,Z 351.274,A -85,B 0,C 180,E1 -13338.092,E2 -13338.092} C_VEL
LIN {X 0,Y 354.808,Z 351.288,A -85,B 0,C 180,E1 -13342.108,E2 -13342.108} C_VEL
LIN {X 0,Y 354.891,Z 351.275,A -85,B 0,C 180,E1 -13345.828,E2 -13345.828} C_VEL
LIN {X 0,Y 354.811,Z 351.289,A -85,B 0,C 180,E1 -13349.683,E2 -13349.683} C_VEL
LIN {X 0,Y 354.801,Z 351.288,A -85,B 0,C 180,E1 -13353.703,E2 -13353.703} C_VEL
LIN {X 0,Y 354.79,Z 351.293,A -85,B 0,C 180,E1 -13356.461,E2 -13356.461} C_VEL
LIN {X 0,Y 354.763,Z 351.297,A -85,B 0,C 180,E1 -13359.413,E2 -13359.413} C_VEL
LIN {X 0,Y 354.82,Z 351.521,A -85,B 0,C 180,E1 -13362.621,E2 -13362.621} C_VEL
LIN {X 0,Y 356.111,Z 357.381,A -85,B 0,C 180,E1 -13365.824,E2 -13365.824} C_VEL
LIN {X 0,Y 357.401,Z 363.921,A -85,B 0,C 180,E1 -13368.983,E2 -13368.983} C_VEL
LIN {X 0,Y 358.641,Z 371.196,A -85,B 0,C 180,E1 -13372.128,E2 -13372.128} C_VEL
LIN {X 0,Y 358.327,Z 374.841,A -85,B 0,C 180,E1 -13373.528,E2 -13373.528} C_VEL
LIN {X 0,Y 356.972,Z 385.099,A -85,B 0,C 180,E1 -13377.221,E2 -13377.221} C_VEL
LIN {X 0,Y 355.902,Z 396.326,A -85,B 0,C 180,E1 -13381.067,E2 -13381.067} C_VEL
LIN {X 0,Y 355.025,Z 407.762,A -85,B 0,C 180,E1 -13384.811,E2 -13384.811} C_VEL
LIN {X 0,Y 354.433,Z 418.866,A -85,B 0,C 180,E1 -13388.282,E2 -13388.282} C_VEL
LIN {X 0,Y 354.656,Z 420.854,A -85,B 0,C 180,E1 -13388.441,E2 -13388.441} C_VEL
LIN {X 0,Y 356.967,Z 433.649,A -85,B 0,C 180,E1 -13389.136,E2 -13389.136} C_VEL
LIN {X 0,Y 358.277,Z 446.853,A -85,B 0,C 180,E1 -13389.983,E2 -13389.983} C_VEL
LIN {X 0,Y 358.595,Z 460.095,A -85,B 0,C 180,E1 -13391.003,E2 -13391.003} C_VEL
